C09106=1048.960,293.791,392.454,172.362,38.885,157.388
C09107=1048.967,294.039,392.422,172.365,38.887,157.388
C09108=1048.973,294.287,392.390,172.369,38.891,157.389
C09109=1048.980,294.535,392.357,172.372,38.894,157.390
C09110=1048.986,294.783,392.325,172.375,38.897,157.391
C09111=1048.993,295.030,392.293,172.379,38.900,157.392
C09112=1048.999,295.279,392.261,172.382,38.903,157.392
C09113=1049.006,295.526,392.229,172.385,38.906,157.393
C09114=1049.012,295.774,392.197,172.389,38.910,157.394
C09115=1049.019,296.021,392.165,172.392,38.913,157.395
C09116=1049.026,296.270,392.132,172.396,38.916,157.396
C09117=1049.032,296.518,392.100,172.398,38.919,157.396
C09118=1049.039,296.765,392.067,172.402,38.923,157.397
C09119=1049.046,297.013,392.035,172.406,38.925,157.398
C09120=1049.052,297.260,392.002,172.408,38.929,157.399
C09121=1049.058,297.509,391.970,172.412,38.932,157.400
C09122=1049.064,297.756,391.937,172.416,38.936,157.401
C09123=1049.071,298.003,391.905,172.419,38.939,157.401
C09124=1049.078,298.252,391.872,172.423,38.942,157.402
C09125=1049.084,298.499,391.839,172.425,38.945,157.403
C09126=1049.090,298.748,391.807,172.429,38.949,157.404
C09127=1049.097,298.995,391.774,172.433,38.952,157.405
C09128=1049.104,299.242,391.742,172.435,38.955,157.405
C09129=1049.110,299.490,391.710,172.439,38.959,157.406
C09130=1049.117,299.738,391.676,172.443,38.961,157.407
C09131=1049.123,299.986,391.644,172.446,38.965,157.408
C09132=1049.129,300.233,391.611,172.449,38.968,157.409
C09133=1049.136,300.481,391.579,172.453,38.971,157.410
C09134=1049.143,300.729,391.546,172.457,38.975,157.410
C09135=1049.150,300.977,391.513,172.460,38.978,157.411
C09136=1049.156,301.224,391.480,172.464,38.982,157.412
C09137=1049.162,301.472,391.447,172.467,38.984,157.413
C09138=1049.169,301.720,391.414,172.470,38.988,157.414
C09139=1049.176,301.967,391.382,172.474,38.991,157.414
C09140=1049.182,302.215,391.349,172.478,38.994,157.415
C09141=1049.189,302.463,391.317,172.481,38.998,157.416
C09142=1049.196,302.711,391.284,172.484,39.001,157.417
C09143=1049.202,302.958,391.251,172.488,39.004,157.418
C09144=1049.208,303.206,391.218,172.492,39.008,157.419
C09145=1049.216,303.454,391.186,172.494,39.011,157.419
C09146=1049.222,303.702,391.153,172.498,39.014,157.420
C09147=1049.229,303.949,391.119,172.502,39.017,157.421
C09148=1049.236,304.197,391.086,172.506,39.021,157.422
C09149=1049.244,304.491,391.047,172.510,39.024,157.423
C09150=1049.251,304.784,391.009,172.513,39.028,157.424
C09151=1049.259,305.078,390.970,172.518,39.032,157.425
C09152=1049.267,305.373,390.930,172.522,39.036,157.426
C09153=1049.274,305.620,390.898,172.526,39.040,157.427
C09154=1049.281,305.867,390.865,172.529,39.043,157.428
C09155=1049.288,306.115,390.831,172.533,39.046,157.428
C09156=1049.294,306.363,390.798,172.536,39.050,157.429
C09157=1049.301,306.611,390.765,172.540,39.053,157.430
C09158=1049.307,306.858,390.732,172.544,39.056,157.431
C09159=1049.314,307.106,390.699,172.547,39.060,157.432
C09160=1049.321,307.354,390.666,172.551,39.063,157.433
C09161=1049.328,307.601,390.632,172.554,39.066,157.434
C09162=1049.335,307.849,390.600,172.558,39.070,157.434
C09163=1049.342,308.096,390.566,172.562,39.073,157.435
C09164=1049.348,308.344,390.533,172.566,39.076,157.436
C09165=1049.355,308.592,390.500,172.568,39.080,157.437
C09166=1049.362,308.839,390.467,172.572,39.083,157.438
C09167=1049.369,309.088,390.434,172.576,39.086,157.439
C09168=1049.375,309.335,390.400,172.580,39.090,157.440
C09169=1049.382,309.583,390.367,172.584,39.093,157.440
C09170=1049.389,309.830,390.334,172.587,39.096,157.441
C09171=1049.396,310.078,390.301,172.591,39.100,157.442
C09172=1049.403,310.325,390.268,172.594,39.103,157.443
C09173=1049.410,310.573,390.235,172.598,39.106,157.444
C09174=1049.417,310.821,390.201,172.602,39.110,157.445
C09175=1049.424,311.068,390.167,172.605,39.113,157.445
C09176=1049.431,311.316,390.134,172.609,39.116,157.446
C09177=1049.437,311.563,390.101,172.613,39.119,157.447
C09178=1049.444,311.811,390.068,172.617,39.123,157.448
C09179=1049.451,312.059,390.034,172.621,39.126,157.449
C09180=1049.458,312.306,390.000,172.624,39.129,157.450
C09181=1049.465,312.554,389.967,172.628,39.133,157.451
C09182=1049.472,312.802,389.933,172.631,39.137,157.452
C09183=1049.479,313.049,389.900,172.635,39.140,157.452
C09184=1049.485,313.297,389.866,172.639,39.143,157.453
C09185=1049.492,313.545,389.832,172.643,39.147,157.454
C09186=1049.499,313.792,389.799,172.646,39.150,157.455
C09187=1049.505,314.040,389.765,172.650,39.154,157.456
C09188=1049.512,314.287,389.731,172.654,39.158,157.457
C09189=1049.518,314.535,389.697,172.658,39.161,157.458
C09190=1049.525,314.783,389.663,172.661,39.164,157.459
C09191=1049.531,315.030,389.629,172.665,39.168,157.460
C09192=1049.538,315.278,389.595,172.669,39.172,157.461
C09193=1049.544,315.525,389.561,172.672,39.175,157.462
C09194=1049.551,315.773,389.527,172.676,39.179,157.462
C09195=1049.558,316.021,389.493,172.680,39.183,157.463
C09196=1049.565,316.268,389.459,172.684,39.186,157.464
C09197=1049.571,316.516,389.425,172.688,39.189,157.465
C09198=1049.578,316.763,389.391,172.692,39.193,157.466
C09199=1049.584,317.011,389.357,172.696,39.196,157.467
C09200=1049.592,317.258,389.322,172.699,39.200,157.468
C09201=1049.598,317.506,389.288,172.703,39.204,157.469
C09202=1049.605,317.753,389.254,172.707,39.207,157.470
C09203=1049.611,318.001,389.220,172.711,39.211,157.471
C09204=1049.618,318.248,389.186,172.714,39.215,157.472
C09205=1049.626,318.546,389.145,172.719,39.219,157.473
C09206=1049.634,318.845,389.103,172.724,39.223,157.474
C09207=1049.642,319.143,389.062,172.728,39.227,157.475
C09208=1049.650,319.441,389.022,172.733,39.232,157.476
C09209=1049.657,319.689,388.986,172.737,39.236,157.477
C09210=1049.664,319.937,388.953,172.741,39.239,157.478
C09211=1049.671,320.185,388.918,172.745,39.243,157.479
C09212=1049.678,320.432,388.884,172.749,39.246,157.480
C09213=1049.684,320.679,388.850,172.753,39.250,157.481
C09214=1049.691,320.927,388.815,172.756,39.253,157.482
C09215=1049.698,321.174,388.781,172.760,39.257,157.483
C09216=1049.705,321.422,388.746,172.764,39.260,157.484
C09217=1049.712,321.670,388.712,172.768,39.264,157.485
C09218=1049.719,321.917,388.677,172.772,39.268,157.486
C09219=1049.726,322.165,388.643,172.776,39.271,157.486
C09220=1049.733,322.412,388.608,172.780,39.275,157.487
C09221=1049.739,322.660,388.574,172.784,39.279,157.488
C09222=1049.746,322.906,388.540,172.788,39.282,157.489
C09223=1049.752,323.154,388.505,172.792,39.286,157.490
C09224=1049.760,323.401,388.471,172.795,39.290,157.491
C09225=1049.766,323.649,388.436,172.799,39.293,157.492
C09226=1049.773,323.897,388.401,172.803,39.297,157.493
C09227=1049.780,324.144,388.367,172.807,39.301,157.494
C09228=1049.787,324.392,388.332,172.811,39.304,157.495
C09229=1049.794,324.639,388.298,172.816,39.308,157.496
C09230=1049.801,324.887,388.263,172.820,39.312,157.497
C09231=1049.808,325.134,388.228,172.824,39.315,157.498
C09232=1049.815,325.382,388.194,172.828,39.319,157.499
C09233=1049.822,325.630,388.159,172.832,39.323,157.500
C09234=1049.830,325.877,388.124,172.836,39.326,157.501
C09235=1049.836,326.125,388.090,172.840,39.330,157.502
C09236=1049.843,326.372,388.055,172.844,39.334,157.503
C09237=1049.851,326.619,388.020,172.847,39.337,157.504
C09238=1049.857,326.867,387.986,172.852,39.341,157.505
C09239=1049.864,327.115,387.951,172.856,39.345,157.506
C09240=1049.871,327.362,387.916,172.860,39.349,157.507
C09241=1049.878,327.609,387.881,172.864,39.352,157.508
C09242=1049.886,327.856,387.846,172.868,39.356,157.509
C09243=1049.893,328.105,387.812,172.872,39.360,157.510
C09244=1049.900,328.352,387.776,172.876,39.364,157.511
C09245=1049.907,328.599,387.742,172.881,39.367,157.512
C09246=1049.914,328.847,387.707,172.885,39.371,157.513
C09247=1049.921,329.094,387.672,172.889,39.375,157.514
C09248=1049.929,329.342,387.637,172.893,39.378,157.515
C09249=1049.935,329.589,387.602,172.897,39.382,157.516
C09250=1049.942,329.836,387.566,172.902,39.386,157.517
C09251=1049.949,330.084,387.531,172.906,39.390,157.518
C09252=1049.956,330.331,387.496,172.910,39.394,157.519
C09253=1049.963,330.579,387.461,172.914,39.398,157.520
C09254=1049.970,330.827,387.426,172.918,39.401,157.521
C09255=1049.977,331.074,387.390,172.922,39.405,157.522
C09256=1049.983,331.321,387.355,172.926,39.409,157.523
C09257=1049.991,331.568,387.319,172.931,39.413,157.524
C09258=1049.997,331.815,387.284,172.935,39.417,157.525
C09259=1050.005,332.064,387.249,172.939,39.421,157.526
C09260=1050.011,332.311,387.214,172.943,39.425,157.527
C09261=1050.019,332.604,387.171,172.948,39.429,157.528
C09262=1050.028,332.897,387.130,172.953,39.434,157.529
C09263=1050.036,333.191,387.087,172.958,39.439,157.530
C09264=1050.044,333.483,387.045,172.963,39.443,157.532
C09265=1050.051,333.731,387.010,172.967,39.447,157.533
C09266=1050.058,333.978,386.975,172.971,39.451,157.534
C09267=1050.066,334.225,386.939,172.975,39.456,157.535
C09268=1050.072,334.473,386.904,172.980,39.459,157.536
C09269=1050.079,334.720,386.868,172.984,39.463,157.537
C09270=1050.086,334.968,386.832,172.988,39.467,157.538
C09271=1050.093,335.215,386.796,172.992,39.471,157.539
C09272=1050.100,335.462,386.761,172.997,39.475,157.540
C09273=1050.107,335.710,386.725,173.001,39.479,157.541
C09274=1050.114,335.957,386.689,173.005,39.483,157.542
C09275=1050.122,336.205,386.654,173.011,39.487,157.543
C09276=1050.129,336.452,386.618,173.015,39.491,157.544
C09277=1050.135,336.699,386.582,173.019,39.495,157.546
C09278=1050.143,336.947,386.546,173.023,39.499,157.547
C09279=1050.150,337.194,386.510,173.028,39.503,157.548
C09280=1050.156,337.441,386.474,173.032,39.507,157.549
C09281=1050.163,337.689,386.438,173.036,39.511,157.550
C09282=1050.170,337.935,386.402,173.041,39.515,157.551
C09283=1050.177,338.184,386.366,173.045,39.519,157.552
C09284=1050.184,338.431,386.330,173.049,39.524,157.553
C09285=1050.192,338.678,386.294,173.054,39.527,157.554
C09286=1050.198,338.925,386.258,173.058,39.532,157.555
C09287=1050.205,339.172,386.223,173.062,39.536,157.556
C09288=1050.213,339.420,386.186,173.067,39.540,157.557
C09289=1050.219,339.667,386.150,173.071,39.544,157.558
C09290=1050.227,339.914,386.114,173.075,39.548,157.560
C09291=1050.234,340.161,386.078,173.081,39.552,157.561
C09292=1050.241,340.409,386.041,173.085,39.556,157.562
C09293=1050.247,340.656,386.006,173.089,39.561,157.563
C09294=1050.255,340.904,385.970,173.094,39.564,157.564
C09295=1050.261,341.151,385.933,173.098,39.569,157.565
C09296=1050.269,341.398,385.897,173.102,39.573,157.566
C09297=1050.277,341.646,385.861,173.107,39.577,157.567
C09298=1050.283,341.893,385.824,173.111,39.581,157.569
C09299=1050.291,342.140,385.788,173.116,39.585,157.570
C09300=1050.298,342.387,385.752,173.120,39.589,157.571
C09301=1050.305,342.635,385.715,173.124,39.594,157.572
C09302=1050.312,342.882,385.679,173.130,39.598,157.573
C09303=1050.319,343.128,385.642,173.134,39.602,157.574
C09304=1050.326,343.376,385.605,173.139,39.607,157.575
C09305=1050.333,343.623,385.569,173.143,39.610,157.576
C09306=1050.340,343.871,385.533,173.148,39.615,157.578
C09307=1050.348,344.118,385.496,173.152,39.619,157.579
C09308=1050.354,344.365,385.460,173.156,39.623,157.580
C09309=1050.361,344.612,385.422,173.161,39.628,157.581
C09310=1050.368,344.859,385.387,173.166,39.632,157.582
C09311=1050.375,345.107,385.350,173.171,39.636,157.583
C09312=1050.383,345.354,385.313,173.175,39.641,157.585
C09313=1050.390,345.601,385.276,173.180,39.645,157.586
C09314=1050.397,345.849,385.240,173.184,39.649,157.587
C09315=1050.405,346.095,385.203,173.189,39.654,157.588
C09316=1050.411,346.343,385.166,173.194,39.658,157.589
C09317=1050.419,346.632,385.123,173.199,39.663,157.591
C09318=1050.428,346.921,385.080,173.204,39.668,157.592
C09319=1050.437,347.211,385.037,173.210,39.673,157.593
C09320=1050.445,347.499,384.994,173.215,39.678,157.595
C09321=1050.452,347.747,384.957,173.220,39.682,157.596
C09322=1050.459,347.994,384.919,173.224,39.687,157.597
C09323=1050.467,348.242,384.883,173.230,39.692,157.598
C09324=1050.473,348.488,384.846,173.234,39.696,157.600
C09325=1050.480,348.735,384.808,173.239,39.700,157.601
C09326=1050.488,348.983,384.772,173.243,39.705,157.602
C09327=1050.495,349.230,384.735,173.248,39.709,157.603
C09328=1050.503,349.477,384.697,173.254,39.714,157.604
C09329=1050.510,349.725,384.660,173.258,39.718,157.606
C09330=1050.517,349.971,384.624,173.263,39.722,157.607
C09331=1050.524,350.218,384.586,173.267,39.727,157.608
C09332=1050.531,350.466,384.549,173.272,39.731,157.609
C09333=1050.538,350.713,384.512,173.277,39.736,157.610
C09334=1050.546,350.960,384.474,173.282,39.740,157.612
C09335=1050.554,351.207,384.437,173.287,39.745,157.613
C09336=1050.561,351.454,384.400,173.291,39.749,157.614
C09337=1050.568,351.701,384.362,173.296,39.754,157.615
C09338=1050.575,351.948,384.325,173.301,39.758,157.617
C09339=1050.582,352.195,384.288,173.306,39.763,157.618
C09340=1050.589,352.442,384.250,173.310,39.768,157.619
C09341=1050.596,352.690,384.213,173.315,39.772,157.620
C09342=1050.604,352.936,384.175,173.321,39.777,157.622
C09343=1050.611,353.183,384.137,173.325,39.781,157.623
C09344=1050.618,353.430,384.100,173.330,39.786,157.624
C09345=1050.625,353.677,384.062,173.336,39.790,157.625
C09346=1050.633,353.925,384.025,173.340,39.795,157.627
C09347=1050.640,354.172,383.987,173.345,39.799,157.628
C09348=1050.647,354.419,383.950,173.349,39.804,157.629
C09349=1050.654,354.666,383.912,173.355,39.809,157.631
C09350=1050.662,354.913,383.875,173.360,39.813,157.632
C09351=1050.669,355.160,383.837,173.364,39.818,157.633
C09352=1050.676,355.407,383.799,173.370,39.823,157.634
C09353=1050.684,355.654,383.761,173.375,39.827,157.636
C09354=1050.691,355.901,383.724,173.379,39.832,157.637
C09355=1050.698,356.148,383.686,173.384,39.837,157.638
C09356=1050.706,356.395,383.648,173.390,39.841,157.639
C09357=1050.714,356.643,383.610,173.395,39.846,157.641
C09358=1050.721,356.889,383.572,173.399,39.851,157.642
C09359=1050.728,357.136,383.535,173.405,39.856,157.643
C09360=1050.736,357.383,383.497,173.410,39.860,157.645
C09361=1050.743,357.630,383.459,173.414,39.865,157.646
C09362=1050.750,357.877,383.421,173.420,39.870,157.647
C09363=1050.757,358.124,383.382,173.425,39.874,157.649
C09364=1050.765,358.372,383.345,173.430,39.879,157.650
C09365=1050.773,358.618,383.306,173.435,39.884,157.651
C09366=1050.780,358.865,383.269,173.440,39.889,157.653
C09367=1050.787,359.112,383.230,173.445,39.894,157.654
C09368=1050.794,359.359,383.192,173.451,39.898,157.655
C09369=1050.801,359.606,383.154,173.455,39.903,157.657
C09370=1050.810,359.853,383.116,173.460,39.908,157.658
C09371=1050.817,360.099,383.077,173.466,39.913,157.659
C09372=1050.824,360.347,383.039,173.471,39.918,157.661
C09373=1050.833,360.641,382.993,173.477,39.924,157.662
C09374=1050.842,360.936,382.948,173.483,39.930,157.664
C09375=1050.851,361.230,382.902,173.489,39.935,157.666
C09376=1050.860,361.525,382.856,173.496,39.941,157.667
C09377=1050.867,361.771,382.818,173.501,39.946,157.669
C09378=1050.874,362.019,382.779,173.506,39.951,157.670
C09379=1050.882,362.266,382.741,173.511,39.956,157.671
C09380=1050.890,362.512,382.703,173.516,39.961,157.673
C09381=1050.897,362.760,382.664,173.522,39.966,157.674
C09382=1050.904,363.006,382.626,173.527,39.971,157.675
C09383=1050.912,363.253,382.587,173.533,39.976,157.677
C09384=1050.919,363.500,382.548,173.537,39.981,157.678
C09385=1050.927,363.747,382.510,173.543,39.986,157.680
C09386=1050.934,363.994,382.471,173.548,39.991,157.681
C09387=1050.942,364.240,382.432,173.553,39.996,157.683
C09388=1050.949,364.487,382.393,173.559,40.001,157.684
C09389=1050.957,364.734,382.355,173.564,40.006,157.685
C09390=1050.964,364.981,382.315,173.570,40.011,157.687
C09391=1050.971,365.228,382.277,173.575,40.016,157.688
C09392=1050.979,365.475,382.237,173.580,40.021,157.690
C09393=1050.986,365.721,382.198,173.585,40.027,157.691
C09394=1050.994,365.969,382.160,173.591,40.032,157.693
C09395=1051.001,366.216,382.121,173.596,40.037,157.694
C09396=1051.009,366.461,382.082,173.602,40.042,157.695
C09397=1051.016,366.709,382.043,173.607,40.047,157.697
C09398=1051.024,366.955,382.005,173.613,40.052,157.698
C09399=1051.032,367.202,381.965,173.618,40.058,157.700
C09400=1051.038,367.449,381.926,173.624,40.063,157.701
C09401=1051.047,367.696,381.886,173.629,40.068,157.703
C09402=1051.054,367.943,381.847,173.635,40.073,157.704
C09403=1051.062,368.189,381.808,173.640,40.078,157.706
C09404=1051.070,368.437,381.769,173.646,40.084,157.707
C09405=1051.077,368.683,381.730,173.651,40.089,157.709
C09406=1051.085,368.930,381.691,173.657,40.094,157.710
C09407=1051.092,369.176,381.651,173.662,40.099,157.712
C09408=1051.100,369.423,381.612,173.668,40.104,157.713
C09409=1051.108,369.670,381.573,173.673,40.110,157.715
C09410=1051.115,369.917,381.533,173.679,40.115,157.716
C09411=1051.123,370.163,381.494,173.684,40.120,157.718
C09412=1051.131,370.411,381.455,173.690,40.125,157.719
C09413=1051.139,370.657,381.416,173.696,40.131,157.721
C09414=1051.146,370.904,381.376,173.701,40.136,157.722
C09415=1051.154,371.150,381.336,173.707,40.141,157.724
C09416=1051.162,371.398,381.297,173.712,40.147,157.725
C09417=1051.169,371.644,381.258,173.718,40.153,157.727
C09418=1051.177,371.891,381.218,173.724,40.158,157.728
C09419=1051.185,372.138,381.178,173.729,40.163,157.730
C09420=1051.192,372.384,381.138,173.735,40.168,157.731
C09421=1051.200,372.631,381.098,173.740,40.174,157.733
C09422=1051.207,372.878,381.059,173.746,40.180,157.734
C09423=1051.214,373.124,381.019,173.753,40.185,157.736
C09424=1051.223,373.371,380.980,173.758,40.191,157.738
C09425=1051.231,373.617,380.940,173.764,40.196,157.739
C09426=1051.239,373.864,380.899,173.770,40.202,157.741
C09427=1051.246,374.111,380.859,173.775,40.207,157.742
C09428=1051.254,374.357,380.820,173.781,40.213,157.744
C09429=1051.264,374.670,380.768,173.788,40.220,157.746
C09430=1051.273,374.985,380.718,173.796,40.227,157.748
C09431=1051.283,375.297,380.667,173.803,40.234,157.750
C09432=1051.293,375.611,380.616,173.810,40.241,157.752
C09433=1051.301,375.858,380.576,173.816,40.247,157.754
C09434=1051.308,376.105,380.536,173.823,40.252,157.755
C09435=1051.317,376.351,380.495,173.828,40.258,157.757
C09436=1051.324,376.598,380.455,173.834,40.264,157.758
C09437=1051.332,376.844,380.415,173.840,40.269,157.760
C09438=1051.340,377.091,380.375,173.846,40.275,157.762
C09439=1051.348,377.337,380.334,173.852,40.280,157.763
C09440=1051.356,377.584,380.294,173.858,40.286,157.765
C09441=1051.363,377.830,380.254,173.864,40.292,157.767
C09442=1051.371,378.077,380.214,173.870,40.298,157.768
C09443=1051.379,378.324,380.173,173.876,40.304,157.770
C09444=1051.387,378.571,380.133,173.882,40.309,157.772
C09445=1051.395,378.817,380.093,173.888,40.315,157.773
C09446=1051.403,379.063,380.052,173.893,40.320,157.775
C09447=1051.411,379.310,380.012,173.900,40.326,157.777
C09448=1051.419,379.556,379.971,173.906,40.332,157.778
C09449=1051.427,379.803,379.931,173.912,40.338,157.780
C09450=1051.435,380.049,379.890,173.919,40.344,157.782
C09451=1051.443,380.295,379.850,173.924,40.350,157.783
C09452=1051.450,380.542,379.809,173.930,40.356,157.785
C09453=1051.458,380.789,379.768,173.936,40.361,157.787
C09454=1051.466,381.035,379.728,173.943,40.368,157.789
C09455=1051.473,381.282,379.687,173.949,40.374,157.790
C09456=1051.482,381.529,379.646,173.954,40.379,157.792
C09457=1051.490,381.775,379.605,173.961,40.386,157.794
C09458=1051.498,382.021,379.563,173.967,40.391,157.795
C09459=1051.506,382.267,379.522,173.973,40.397,157.797
C09460=1051.514,382.513,379.482,173.980,40.403,157.799
C09461=1051.521,382.760,379.440,173.986,40.409,157.801
C09462=1051.530,383.007,379.399,173.992,40.416,157.802
C09463=1051.538,383.253,379.359,173.998,40.421,157.804
C09464=1051.545,383.500,379.318,174.004,40.428,157.806
C09465=1051.553,383.746,379.276,174.011,40.433,157.808
C09466=1051.561,383.992,379.236,174.017,40.440,157.809
C09467=1051.569,384.239,379.194,174.024,40.446,157.811
C09468=1051.578,384.485,379.153,174.030,40.452,157.813
C09469=1051.586,384.731,379.112,174.036,40.458,157.815
C09470=1051.593,384.978,379.070,174.043,40.464,157.817
C09471=1051.602,385.224,379.029,174.049,40.471,157.818
C09472=1051.610,385.470,378.988,174.056,40.476,157.820
C09473=1051.618,385.717,378.946,174.062,40.483,157.822
C09474=1051.626,385.963,378.906,174.069,40.489,157.824
C09475=1051.634,386.210,378.863,174.075,40.495,157.826
C09476=1051.642,386.456,378.823,174.082,40.501,157.828
C09477=1051.651,386.702,378.781,174.087,40.508,157.829
C09478=1051.659,386.949,378.739,174.094,40.514,157.831
C09479=1051.667,387.195,378.698,174.100,40.520,157.833
C09480=1051.675,387.442,378.656,174.107,40.526,157.835
C09481=1051.683,387.687,378.615,174.113,40.533,157.837
C09482=1051.692,387.934,378.574,174.120,40.539,157.839
C09483=1051.700,388.180,378.532,174.126,40.545,157.840
C09484=1051.708,388.427,378.490,174.133,40.551,157.842
C09485=1051.719,388.772,378.432,174.142,40.560,157.845
C09486=1051.732,389.118,378.373,174.152,40.569,157.848
C09487=1051.743,389.465,378.314,174.161,40.578,157.850
C09488=1051.755,389.810,378.256,174.171,40.587,157.853
C09489=1051.763,390.056,378.213,174.177,40.594,157.855
C09490=1051.771,390.303,378.171,174.184,40.600,157.857
C09491=1051.779,390.549,378.130,174.191,40.607,157.859
C09492=1051.788,390.795,378.087,174.197,40.613,157.861
C09493=1051.795,391.041,378.045,174.204,40.620,157.862
C09494=1051.804,391.288,378.004,174.211,40.626,157.865
C09495=1051.813,391.534,377.961,174.218,40.633,157.866
C09496=1051.820,391.780,377.919,174.225,40.639,157.868
C09497=1051.829,392.026,377.877,174.232,40.646,157.870
C09498=1051.837,392.273,377.835,174.238,40.653,157.872
C09499=1051.846,392.519,377.792,174.245,40.659,157.874
C09500=1051.853,392.765,377.750,174.252,40.666,157.876
C09501=1051.862,393.011,377.708,174.259,40.673,157.878
C09502=1051.871,393.257,377.665,174.266,40.679,157.880
C09503=1051.878,393.503,377.623,174.273,40.686,157.882
C09504=1051.887,393.749,377.580,174.280,40.693,157.884
C09505=1051.895,393.996,377.538,174.286,40.700,157.886
C09506=1051.904,394.242,377.495,174.293,40.706,157.888
C09507=1051.913,394.488,377.452,174.301,40.713,157.890
C09508=1051.920,394.734,377.410,174.308,40.720,157.892
C09509=1051.929,394.980,377.367,174.315,40.726,157.894
C09510=1051.937,395.226,377.324,174.321,40.734,157.897
C09511=1051.946,395.472,377.282,174.329,40.741,157.899
C09512=1051.954,395.718,377.239,174.336,40.747,157.901
C09513=1051.963,395.965,377.196,174.343,40.754,157.903
C09514=1051.972,396.210,377.153,174.350,40.761,157.905
C09515=1051.980,396.457,377.111,174.358,40.768,157.907
C09516=1051.989,396.703,377.068,174.364,40.775,157.909
C09517=1051.997,396.949,377.025,174.371,40.782,157.911
C09518=1052.006,397.195,376.982,174.378,40.789,157.913
C09519=1052.013,397.441,376.938,174.386,40.796,157.915
C09520=1052.022,397.688,376.895,174.393,40.803,157.917
C09521=1052.030,397.934,376.852,174.400,40.810,157.919
C09522=1052.039,398.180,376.809,174.408,40.817,157.922
C09523=1052.047,398.426,376.766,174.415,40.824,157.924
C09524=1052.056,398.672,376.723,174.423,40.831,157.926
C09525=1052.065,398.917,376.679,174.429,40.838,157.928
C09526=1052.073,399.163,376.636,174.436,40.845,157.930
C09527=1052.082,399.409,376.593,174.444,40.853,157.932
C09528=1052.090,399.655,376.550,174.451,40.860,157.935
C09529=1052.100,399.901,376.506,174.459,40.867,157.937
C09530=1052.108,400.148,376.463,174.466,40.874,157.939
C09531=1052.117,400.394,376.420,174.474,40.881,157.941
C09532=1052.125,400.639,376.376,174.481,40.889,157.943
C09533=1052.133,400.885,376.333,174.488,40.896,157.946
C09534=1052.143,401.132,376.289,174.496,40.903,157.948
C09535=1052.151,401.378,376.246,174.503,40.910,157.950
C09536=1052.160,401.623,376.202,174.511,40.917,157.952
C09537=1052.168,401.870,376.158,174.519,40.925,157.954
C09538=1052.177,402.116,376.114,174.527,40.932,157.957
C09539=1052.186,402.362,376.071,174.534,40.939,157.959
C09540=1052.195,402.608,376.027,174.542,40.947,157.961
C09541=1052.207,402.971,375.962,174.553,40.958,157.964
C09542=1052.221,403.336,375.897,174.564,40.969,157.968
C09543=1052.233,403.700,375.832,174.575,40.980,157.971
C09544=1052.246,404.064,375.767,174.587,40.991,157.975
C09545=1052.255,404.310,375.723,174.595,40.999,157.977
C09546=1052.264,404.556,375.678,174.602,41.007,157.979
C09547=1052.272,404.802,375.635,174.611,41.014,157.982
C09548=1052.282,405.048,375.590,174.618,41.021,157.984
C09549=1052.290,405.294,375.546,174.626,41.029,157.986
C09550=1052.299,405.540,375.501,174.634,41.037,157.989
C09551=1052.307,405.785,375.458,174.641,41.045,157.991
C09552=1052.316,406.032,375.413,174.650,41.052,157.993
C09553=1052.325,406.277,375.368,174.658,41.060,157.996
C09554=1052.334,406.523,375.324,174.666,41.068,157.998
C09555=1052.343,406.769,375.280,174.673,41.076,158.001
C09556=1052.351,407.015,375.235,174.682,41.083,158.003
C09557=1052.360,407.261,375.190,174.690,41.091,158.005
C09558=1052.370,407.507,375.146,174.697,41.099,158.008
C09559=1052.378,407.752,375.101,174.706,41.107,158.010
C09560=1052.388,407.998,375.057,174.714,41.115,158.013
C09561=1052.396,408.244,375.011,174.722,41.123,158.015
C09562=1052.405,408.490,374.967,174.730,41.131,158.018
C09563=1052.414,408.735,374.922,174.738,41.138,158.020
C09564=1052.423,408.982,374.877,174.746,41.147,158.023
C09565=1052.433,409.227,374.833,174.755,41.154,158.025
C09566=1052.441,409.474,374.788,174.763,41.162,158.028
C09567=1052.450,409.719,374.743,174.772,41.170,158.030
C09568=1052.459,409.964,374.698,174.779,41.179,158.033
C09569=1052.468,410.210,374.653,174.787,41.186,158.035
C09570=1052.478,410.456,374.608,174.796,41.194,158.038
C09571=1052.487,410.702,374.563,174.804,41.203,158.040
C09572=1052.496,410.948,374.518,174.813,41.211,158.043
C09573=1052.505,411.194,374.473,174.821,41.219,158.045
C09574=1052.514,411.439,374.427,174.830,41.227,158.048
C09575=1052.523,411.685,374.382,174.839,41.235,158.050
C09576=1052.533,411.931,374.337,174.846,41.243,158.053
C09577=1052.542,412.177,374.292,174.856,41.252,158.056
C09578=1052.552,412.422,374.247,174.863,41.260,158.058
C09579=1052.561,412.668,374.201,174.872,41.268,158.061
C09580=1052.570,412.914,374.156,174.880,41.277,158.064
C09581=1052.580,413.159,374.111,174.889,41.285,158.066
C09582=1052.589,413.404,374.065,174.899,41.293,158.069
C09583=1052.598,413.650,374.020,174.906,41.301,158.071
C09584=1052.607,413.896,373.974,174.916,41.310,158.074
C09585=1052.617,414.142,373.928,174.925,41.318,158.077
C09586=1052.626,414.388,373.882,174.933,41.327,158.079
C09587=1052.635,414.633,373.836,174.942,41.335,158.082
C09588=1052.644,414.879,373.791,174.951,41.344,158.085
C09589=1052.653,415.124,373.745,174.959,41.352,158.088
C09590=1052.663,415.370,373.698,174.968,41.361,158.090
C09591=1052.672,415.616,373.653,174.977,41.369,158.093
C09592=1052.681,415.861,373.607,174.986,41.378,158.096
C09593=1052.691,416.106,373.560,174.995,41.387,158.098
C09594=1052.700,416.353,373.515,175.004,41.395,158.101
C09595=1052.709,416.598,373.469,175.013,41.404,158.104
C09596=1052.719,416.843,373.422,175.022,41.413,158.107
C09597=1052.733,417.218,373.352,175.036,41.426,158.111
C09598=1052.748,417.593,373.281,175.050,41.439,158.115
C09599=1052.762,417.968,373.211,175.064,41.452,158.120
C09600=1052.777,418.341,373.140,175.078,41.466,158.124
C09601=1052.787,418.587,373.093,175.087,41.475,158.127
C09602=1052.796,418.832,373.047,175.097,41.484,158.130
C09603=1052.806,419.078,373.001,175.106,41.493,158.132
C09604=1052.815,419.324,372.955,175.115,41.502,158.135
C09605=1052.825,419.570,372.907,175.125,41.511,158.138
C09606=1052.834,419.814,372.861,175.134,41.520,158.141
C09607=1052.844,420.060,372.814,175.144,41.529,158.144
C09608=1052.854,420.305,372.767,175.153,41.538,158.147
C09609=1052.863,420.551,372.720,175.163,41.547,158.150
C09610=1052.873,420.796,372.673,175.172,41.556,158.153
C09611=1052.882,421.042,372.627,175.181,41.565,158.156
C09612=1052.892,421.287,372.579,175.191,41.575,158.159
C09613=1052.902,421.532,372.532,175.200,41.584,158.162
C09614=1052.911,421.778,372.486,175.210,41.593,158.165
C09615=1052.921,422.023,372.438,175.219,41.602,158.168
C09616=1052.931,422.268,372.391,175.230,41.612,158.171
C09617=1052.941,422.514,372.343,175.240,41.621,158.174
C09618=1052.950,422.759,372.297,175.249,41.630,158.177
C09619=1052.960,423.005,372.249,175.259,41.640,158.180
C09620=1052.970,423.250,372.202,175.268,41.649,158.183
C09621=1052.979,423.493,372.155,175.279,41.658,158.186
C09622=1052.989,423.736,372.108,175.289,41.667,158.189
C09623=1052.999,423.980,372.061,175.298,41.677,158.192
C09624=1053.009,424.223,372.014,175.308,41.686,158.195
C09625=1053.019,424.466,371.967,175.319,41.696,158.199
C09626=1053.030,424.709,371.919,175.328,41.705,158.202
C09627=1053.039,424.952,371.872,175.338,41.715,158.205
C09628=1053.049,425.195,371.826,175.349,41.724,158.208
C09629=1053.058,425.441,371.778,175.358,41.733,158.211
C09630=1053.069,425.686,371.730,175.368,41.743,158.214
C09631=1053.078,425.931,371.682,175.379,41.753,158.218
C09632=1053.089,426.176,371.634,175.389,41.763,158.221
C09633=1053.099,426.422,371.586,175.400,41.773,158.224
C09634=1053.109,426.667,371.538,175.409,41.782,158.227
C09635=1053.119,426.912,371.490,175.420,41.792,158.230
C09636=1053.129,427.157,371.442,175.430,41.802,158.234
C09637=1053.139,427.402,371.394,175.441,41.812,158.237
C09638=1053.148,427.648,371.346,175.451,41.822,158.240
C09639=1053.159,427.892,371.298,175.462,41.831,158.243
C09640=1053.169,428.138,371.249,175.472,41.842,158.247
C09641=1053.179,428.383,371.201,175.483,41.852,158.250
C09642=1053.190,428.628,371.153,175.494,41.861,158.253
C09643=1053.199,428.872,371.104,175.504,41.872,158.257
C09644=1053.210,429.118,371.056,175.515,41.882,158.260
C09645=1053.220,429.363,371.007,175.526,41.891,158.264
C09646=1053.231,429.609,370.958,175.536,41.902,158.267
C09647=1053.241,429.853,370.910,175.547,41.912,158.270
C09648=1053.251,430.098,370.861,175.558,41.922,158.274
C09649=1053.262,430.343,370.812,175.569,41.932,158.277
C09650=1053.271,430.588,370.764,175.579,41.943,158.281
C09651=1053.282,430.833,370.714,175.591,41.953,158.284
C09652=1053.292,431.078,370.666,175.602,41.963,158.288
C09653=1053.309,431.470,370.587,175.619,41.980,158.293
C09654=1053.325,431.864,370.508,175.637,41.997,158.299
C09655=1053.342,432.256,370.430,175.655,42.014,158.305
C09656=1053.359,432.649,370.351,175.673,42.030,158.310
C09657=1053.369,432.894,370.301,175.684,42.041,158.314
C09658=1053.379,433.139,370.252,175.696,42.051,158.318
C09659=1053.390,433.384,370.202,175.707,42.062,158.321
C09660=1053.400,433.628,370.153,175.719,42.073,158.325
C09661=1053.412,433.873,370.104,175.730,42.084,158.329
C09662=1053.422,434.118,370.054,175.741,42.094,158.332
C09663=1053.433,434.363,370.005,175.754,42.105,158.336
C09664=1053.443,434.607,369.955,175.765,42.116,158.340
C09665=1053.454,434.853,369.906,175.777,42.126,158.343
C09666=1053.464,435.098,369.856,175.788,42.137,158.347
C09667=1053.475,435.342,369.806,175.800,42.148,158.351
C09668=1053.486,435.587,369.756,175.811,42.159,158.354
C09669=1053.497,435.832,369.707,175.824,42.170,158.358
C09670=1053.508,436.077,369.656,175.836,42.181,158.362
C09671=1053.518,436.322,369.607,175.847,42.192,158.366
C09672=1053.529,436.566,369.556,175.860,42.202,158.369
C09673=1053.541,436.811,369.507,175.872,42.214,158.373
C09674=1053.551,437.056,369.456,175.883,42.225,158.377
C09675=1053.562,437.300,369.406,175.896,42.236,158.381
C09676=1053.573,437.544,369.356,175.908,42.247,158.385
C09677=1053.583,437.789,369.306,175.920,42.259,158.389
C09678=1053.594,438.034,369.256,175.932,42.270,158.393
C09679=1053.605,438.278,369.206,175.944,42.281,158.397
C09680=1053.617,438.523,369.155,175.957,42.292,158.401
C09681=1053.627,438.768,369.104,175.969,42.304,158.405
C09682=1053.638,439.013,369.054,175.982,42.315,158.409
C09683=1053.649,439.256,369.003,175.994,42.327,158.413
C09684=1053.661,439.502,368.952,176.007,42.338,158.417
C09685=1053.671,439.746,368.901,176.020,42.349,158.421
C09686=1053.683,439.990,368.850,176.032,42.361,158.425
C09687=1053.694,440.234,368.800,176.045,42.372,158.429
C09688=1053.705,440.480,368.749,176.058,42.384,158.433
C09689=1053.716,440.724,368.697,176.070,42.396,158.437
C09690=1053.727,440.969,368.647,176.083,42.407,158.441
C09691=1053.738,441.213,368.596,176.096,42.419,158.445
C09692=1053.749,441.457,368.544,176.109,42.431,158.449
C09693=1053.761,441.702,368.493,176.121,42.443,158.454
C09694=1053.772,441.946,368.442,176.134,42.454,158.458
C09695=1053.783,442.191,368.390,176.148,42.466,158.462
C09696=1053.795,442.435,368.339,176.161,42.478,158.466
C09697=1053.806,442.679,368.288,176.174,42.490,158.471
C09698=1053.817,442.924,368.236,176.188,42.502,158.475
C09699=1053.829,443.168,368.184,176.201,42.514,158.479
C09700=1053.840,443.412,368.133,176.214,42.526,158.483
C09701=1053.852,443.657,368.081,176.228,42.538,158.488
C09702=1053.863,443.901,368.029,176.241,42.550,158.492
C09703=1053.874,444.145,367.978,176.255,42.563,158.496
C09704=1053.886,444.390,367.926,176.268,42.574,158.501
C09705=1053.898,444.634,367.873,176.281,42.587,158.505
C09706=1053.910,444.878,367.822,176.295,42.599,158.510
C09707=1053.921,445.122,367.769,176.310,42.611,158.514
C09708=1053.932,445.366,367.718,176.323,42.624,158.519
C09709=1053.945,445.612,367.666,176.337,42.636,158.523
C09710=1053.956,445.858,367.613,176.351,42.649,158.528
C09711=1053.967,446.104,367.560,176.365,42.661,158.532
C09712=1053.979,446.349,367.508,176.379,42.674,158.537
C09713=1053.992,446.592,367.456,176.394,42.686,158.541
C09714=1054.005,446.835,367.404,176.407,42.698,158.546
C09715=1054.018,447.079,367.354,176.422,42.711,158.550
C09716=1054.032,447.323,367.303,176.436,42.722,158.554
C09717=1054.048,447.567,367.254,176.450,42.734,158.559
C09718=1054.063,447.811,367.204,176.464,42.745,158.563
C09719=1054.080,448.055,367.157,176.480,42.757,158.567
C09720=1054.098,448.300,367.108,176.494,42.768,158.572
C09721=1054.116,448.544,367.060,176.508,42.779,158.576
C09722=1054.134,448.789,367.013,176.523,42.790,158.580
C09723=1054.154,449.034,366.967,176.538,42.800,158.584
C09724=1054.175,449.278,366.921,176.552,42.811,158.588
C09725=1054.196,449.524,366.876,176.568,42.821,158.592
C09726=1054.218,449.769,366.831,176.582,42.831,158.596
C09727=1054.241,450.015,366.787,176.598,42.841,158.600
C09728=1054.264,450.259,366.743,176.613,42.851,158.604
C09729=1053.943,450.280,366.451,176.612,42.951,158.633
C09730=1053.920,450.036,366.495,176.596,42.941,158.629
C09731=1053.897,449.790,366.539,176.582,42.931,158.625
C09732=1053.876,449.545,366.584,176.567,42.921,158.621
C09733=1053.854,449.299,366.629,176.551,42.911,158.617
C09734=1053.833,449.054,366.674,176.536,42.901,158.613
C09735=1053.813,448.810,366.721,176.521,42.890,158.608
C09736=1053.793,448.565,366.768,176.506,42.879,158.604
C09737=1053.776,448.320,366.815,176.492,42.868,158.600
C09738=1053.758,448.076,366.863,176.476,42.857,158.596
C09739=1053.742,447.831,366.912,176.462,42.846,158.591
C09740=1053.725,447.588,366.961,176.448,42.835,158.587
C09741=1053.710,447.344,367.010,176.433,42.823,158.583
C09742=1053.695,447.107,367.059,176.420,42.812,158.579
C09743=1053.682,446.871,367.108,176.405,42.800,158.574
C09744=1053.670,446.635,367.158,176.392,42.788,158.570
C09745=1053.658,446.400,367.208,176.378,42.777,158.566
C09746=1053.646,446.166,367.258,176.365,42.765,158.561
C09747=1053.635,445.932,367.308,176.351,42.752,158.557
C09748=1053.625,445.697,367.359,176.338,42.741,158.552
C09749=1053.613,445.463,367.408,176.324,42.729,158.548
C09750=1053.601,445.218,367.461,176.310,42.717,158.544
C09751=1053.590,444.974,367.512,176.296,42.704,158.539
C09752=1053.577,444.730,367.564,176.283,42.693,158.535
C09753=1053.566,444.486,367.617,176.269,42.680,158.530
C09754=1053.554,444.241,367.669,176.255,42.668,158.526
C09755=1053.543,443.996,367.721,176.241,42.656,158.522
C09756=1053.531,443.753,367.772,176.227,42.644,158.517
C09757=1053.520,443.508,367.824,176.214,42.632,158.513
C09758=1053.508,443.264,367.876,176.201,42.620,158.509
C09759=1053.496,443.019,367.927,176.187,42.608,158.504
C09760=1053.486,442.775,367.979,176.174,42.596,158.500
C09761=1053.474,442.531,368.030,176.161,42.584,158.496
C09762=1053.463,442.287,368.082,176.147,42.572,158.491
C09763=1053.452,442.042,368.133,176.134,42.560,158.487
C09764=1053.440,441.798,368.185,176.122,42.548,158.483
C09765=1053.429,441.553,368.236,176.108,42.537,158.479
C09766=1053.417,441.309,368.288,176.095,42.525,158.475
C09767=1053.406,441.065,368.338,176.082,42.514,158.470
C09768=1053.395,440.820,368.390,176.069,42.502,158.466
C09769=1053.384,440.576,368.441,176.056,42.491,158.462
C09770=1053.373,440.331,368.491,176.044,42.479,158.458
C09771=1053.361,440.087,368.543,176.031,42.467,158.454
C09772=1053.351,439.842,368.594,176.017,42.456,158.450
C09773=1053.340,439.598,368.644,176.006,42.445,158.446
C09774=1053.328,439.353,368.695,175.993,42.433,158.442
C09775=1053.317,439.109,368.746,175.980,42.422,158.438
C09776=1053.307,438.864,368.797,175.968,42.410,158.434
C09777=1053.295,438.619,368.847,175.955,42.399,158.430
C09778=1053.284,438.375,368.898,175.943,42.388,158.426
C09779=1053.273,438.130,368.948,175.930,42.376,158.422
C09780=1053.262,437.886,368.998,175.918,42.365,158.418
C09781=1053.251,437.641,369.049,175.905,42.354,158.414
C09782=1053.240,437.397,369.099,175.894,42.343,158.410
C09783=1053.230,437.152,369.150,175.882,42.332,158.406
C09784=1053.218,436.907,369.201,175.869,42.321,158.403
C09785=1053.208,436.662,369.250,175.857,42.310,158.399
C09786=1053.197,436.417,369.301,175.844,42.299,158.395
C09787=1053.186,436.172,369.350,175.833,42.288,158.391
C09788=1053.175,435.928,369.400,175.821,42.277,158.387
C09789=1053.164,435.683,369.449,175.809,42.266,158.383
C09790=1053.153,435.439,369.500,175.797,42.255,158.380
C09791=1053.142,435.194,369.549,175.785,42.244,158.376
C09792=1053.132,434.950,369.599,175.774,42.234,158.372
C09793=1053.121,434.705,369.649,175.762,42.223,158.369
C09794=1053.110,434.460,369.699,175.750,42.212,158.365
C09795=1053.100,434.215,369.748,175.738,42.202,158.361
C09796=1053.089,433.970,369.798,175.727,42.191,158.357
C09797=1053.078,433.725,369.847,175.715,42.180,158.354
C09798=1053.068,433.480,369.897,175.704,42.169,158.350
C09799=1053.057,433.236,369.946,175.692,42.159,158.346
C09800=1053.046,432.991,369.995,175.681,42.149,158.343
C09801=1053.036,432.746,370.045,175.670,42.138,158.339
C09802=1053.019,432.351,370.124,175.652,42.121,158.334
C09803=1053.002,431.957,370.204,175.633,42.104,158.328
C09804=1052.986,431.562,370.283,175.615,42.088,158.322
C09805=1052.969,431.166,370.362,175.597,42.071,158.316
C09806=1052.959,430.921,370.411,175.586,42.061,158.313
C09807=1052.949,430.676,370.460,175.574,42.050,158.309
C09808=1052.937,430.431,370.509,175.564,42.040,158.306
C09809=1052.928,430.187,370.557,175.553,42.030,158.302
C09810=1052.918,429.942,370.607,175.542,42.019,158.299
C09811=1052.907,429.697,370.655,175.531,42.010,158.296
C09812=1052.897,429.452,370.704,175.521,41.999,158.292
C09813=1052.886,429.206,370.752,175.510,41.989,158.289
C09814=1052.877,428.961,370.801,175.498,41.979,158.285
C09815=1052.866,428.717,370.849,175.487,41.969,158.282
C09816=1052.856,428.471,370.898,175.477,41.959,158.279
C09817=1052.846,428.226,370.946,175.466,41.950,158.275
C09818=1052.836,427.981,370.994,175.455,41.940,158.272
C09819=1052.826,427.736,371.043,175.445,41.929,158.269
C09820=1052.815,427.491,371.091,175.434,41.920,158.265
C09821=1052.805,427.246,371.139,175.425,41.910,158.262
C09822=1052.795,427.000,371.187,175.414,41.900,158.259
C09823=1052.785,426.756,371.235,175.404,41.890,158.256
C09824=1052.775,426.511,371.284,175.393,41.881,158.252
C09825=1052.765,426.265,371.331,175.383,41.871,158.249
C09826=1052.755,426.020,371.380,175.372,41.861,158.246
C09827=1052.744,425.774,371.427,175.362,41.851,158.243
C09828=1052.735,425.529,371.476,175.351,41.842,158.239
C09829=1052.724,425.284,371.523,175.342,41.833,158.236
C09830=1052.715,425.039,371.571,175.331,41.823,158.233
C09831=1052.705,424.794,371.618,175.321,41.813,158.230
C09832=1052.694,424.549,371.666,175.311,41.804,158.227
C09833=1052.685,424.303,371.714,175.301,41.795,158.224
C09834=1052.675,424.058,371.761,175.291,41.785,158.221
C09835=1052.665,423.812,371.808,175.281,41.776,158.217
C09836=1052.655,423.568,371.856,175.271,41.766,158.214
C09837=1052.645,423.322,371.904,175.261,41.757,158.211
C09838=1052.635,423.078,371.951,175.251,41.747,158.208
C09839=1052.626,422.832,371.998,175.241,41.739,158.205
C09840=1052.616,422.586,372.045,175.231,41.729,158.202
C09841=1052.605,422.341,372.092,175.221,41.720,158.199
C09842=1052.596,422.095,372.140,175.212,41.711,158.196
C09843=1052.586,421.851,372.187,175.202,41.701,158.193
C09844=1052.576,421.605,372.234,175.192,41.692,158.190
C09845=1052.567,421.359,372.281,175.182,41.683,158.187
C09846=1052.557,421.114,372.328,175.173,41.674,158.184
C09847=1052.547,420.869,372.375,175.163,41.665,158.181
C09848=1052.537,420.623,372.422,175.154,41.656,158.178
C09849=1052.529,420.379,372.469,175.144,41.646,158.175
C09850=1052.519,420.133,372.516,175.135,41.637,158.172
C09851=1052.508,419.887,372.563,175.125,41.628,158.169
C09852=1052.500,419.642,372.609,175.116,41.619,158.166
C09853=1052.490,419.397,372.657,175.106,41.610,158.163
C09854=1052.480,419.151,372.703,175.097,41.602,158.161
C09855=1052.471,418.905,372.749,175.088,41.593,158.158
C09856=1052.461,418.660,372.795,175.078,41.584,158.155
C09857=1052.451,418.414,372.842,175.069,41.575,158.152
C09858=1052.437,418.041,372.913,175.055,41.562,158.148
C09859=1052.422,417.670,372.982,175.041,41.548,158.143
C09860=1052.408,417.297,373.053,175.027,41.535,158.139
C09861=1052.393,416.924,373.123,175.013,41.522,158.135
C09862=1052.384,416.679,373.170,175.004,41.514,158.132
C09863=1052.375,416.433,373.216,174.994,41.505,158.129
C09864=1052.365,416.187,373.262,174.985,41.496,158.126
C09865=1052.356,415.942,373.308,174.977,41.487,158.124
C09866=1052.346,415.700,373.353,174.968,41.479,158.121
C09867=1052.337,415.459,373.399,174.959,41.471,158.118
C09868=1052.328,415.217,373.443,174.950,41.462,158.116
C09869=1052.319,414.975,373.490,174.941,41.454,158.113
C09870=1052.309,414.733,373.534,174.932,41.446,158.110
C09871=1052.300,414.491,373.579,174.924,41.437,158.107
C09872=1052.291,414.250,373.625,174.915,41.429,158.105
C09873=1052.282,414.008,373.669,174.906,41.420,158.102
C09874=1052.273,413.762,373.715,174.898,41.412,158.100
C09875=1052.264,413.517,373.761,174.889,41.404,158.097
C09876=1052.255,413.271,373.806,174.880,41.396,158.094
C09877=1052.245,413.025,373.852,174.872,41.387,158.092
C09878=1052.236,412.779,373.898,174.863,41.379,158.089
C09879=1052.226,412.534,373.943,174.854,41.371,158.086
C09880=1052.217,412.288,373.988,174.846,41.362,158.084
C09881=1052.208,412.042,374.034,174.837,41.354,158.081
C09882=1052.198,411.797,374.078,174.829,41.346,158.079
C09883=1052.189,411.551,374.124,174.820,41.338,158.076
C09884=1052.180,411.305,374.169,174.812,41.330,158.073
C09885=1052.171,411.060,374.214,174.803,41.322,158.071
C09886=1052.162,410.814,374.260,174.795,41.314,158.068
C09887=1052.152,410.568,374.304,174.786,41.306,158.066
C09888=1052.143,410.322,374.350,174.778,41.297,158.063
C09889=1052.134,410.076,374.395,174.769,41.290,158.061
C09890=1052.125,409.831,374.439,174.762,41.282,158.058
C09891=1052.116,409.585,374.485,174.753,41.274,158.056
C09892=1052.107,409.340,374.529,174.745,41.266,158.053
C09893=1052.098,409.093,374.574,174.736,41.258,158.051
C09894=1052.089,408.848,374.619,174.728,41.250,158.048
C09895=1052.079,408.602,374.664,174.719,41.242,158.046
C09896=1052.071,408.356,374.709,174.711,41.234,158.043
C09897=1052.061,408.111,374.753,174.704,41.226,158.041
C09898=1052.053,407.864,374.798,174.695,41.218,158.038
C09899=1052.044,407.619,374.843,174.687,41.211,158.036
C09900=1052.034,407.372,374.888,174.679,41.203,158.034
C09901=1052.026,407.127,374.933,174.670,41.195,158.031
C09902=1052.017,406.881,374.977,174.663,41.187,158.029
C09903=1052.009,406.635,375.021,174.655,41.180,158.026
C09904=1051.999,406.390,375.066,174.646,41.172,158.024
C09905=1051.990,406.143,375.111,174.639,41.164,158.021
C09906=1051.982,405.898,375.155,174.631,41.157,158.019
C09907=1051.973,405.652,375.199,174.623,41.149,158.017
C09908=1051.965,405.406,375.243,174.615,41.141,158.014
C09909=1051.955,405.160,375.288,174.607,41.134,158.012
C09910=1051.947,404.915,375.333,174.599,41.126,158.010
C09911=1051.937,404.668,375.377,174.591,41.118,158.007
C09912=1051.929,404.423,375.421,174.584,41.111,158.005
C09913=1051.920,404.177,375.465,174.575,41.104,158.003
C09914=1051.907,403.802,375.532,174.564,41.092,157.999
C09915=1051.894,403.429,375.598,174.552,41.080,157.995
C09916=1051.880,403.055,375.666,174.540,41.069,157.992
C09917=1051.867,402.681,375.732,174.528,41.058,157.989
C09918=1051.858,402.436,375.776,174.521,41.051,157.986
C09919=1051.849,402.189,375.819,174.513,41.044,157.984
C09920=1051.841,401.943,375.864,174.506,41.036,157.982
C09921=1051.832,401.698,375.907,174.498,41.029,157.980
C09922=1051.823,401.451,375.951,174.491,41.022,157.977
C09923=1051.814,401.206,375.995,174.483,41.014,157.975
C09924=1051.806,400.960,376.038,174.476,41.007,157.973
C09925=1051.796,400.713,376.082,174.468,41.000,157.971
C09926=1051.789,400.467,376.125,174.461,40.993,157.969
C09927=1051.780,400.221,376.168,174.454,40.986,157.966
C09928=1051.771,399.976,376.212,174.446,40.978,157.964
C09929=1051.762,399.729,376.255,174.439,40.971,157.962
C09930=1051.754,399.483,376.299,174.431,40.964,157.960
C09931=1051.745,399.237,376.342,174.424,40.957,157.958
C09932=1051.736,398.991,376.385,174.416,40.950,157.955
C09933=1051.728,398.745,376.428,174.409,40.943,157.953
C09934=1051.719,398.499,376.471,174.402,40.936,157.951
C09935=1051.711,398.254,376.515,174.394,40.928,157.949
C09936=1051.702,398.008,376.558,174.387,40.922,157.947
C09937=1051.693,397.761,376.601,174.379,40.915,157.945
C09938=1051.685,397.515,376.645,174.372,40.907,157.942
C09939=1051.677,397.268,376.688,174.365,40.901,157.940
C09940=1051.668,397.022,376.731,174.357,40.893,157.938
C09941=1051.660,396.776,376.774,174.350,40.887,157.936
C09942=1051.652,396.531,376.817,174.344,40.880,157.934
C09943=1051.643,396.284,376.860,174.336,40.873,157.932
C09944=1051.634,396.038,376.902,174.329,40.866,157.930
C09945=1051.626,395.793,376.945,174.322,40.859,157.928
C09946=1051.617,395.547,376.988,174.314,40.852,157.926
C09947=1051.609,395.300,377.031,174.307,40.845,157.924
C09948=1051.601,395.054,377.073,174.300,40.839,157.922
C09949=1051.592,394.808,377.116,174.294,40.832,157.920
C09950=1051.584,394.562,377.159,174.286,40.825,157.918
C09951=1051.575,394.315,377.201,174.279,40.819,157.916
C09952=1051.566,394.069,377.244,174.272,40.812,157.914
C09953=1051.558,393.824,377.286,174.266,40.805,157.912
C09954=1051.550,393.577,377.329,174.258,40.798,157.910
C09955=1051.542,393.331,377.372,174.251,40.792,157.907
C09956=1051.534,393.085,377.414,174.244,40.785,157.905
C09957=1051.525,392.839,377.456,174.238,40.778,157.903
C09958=1051.517,392.593,377.498,174.231,40.772,157.902
C09959=1051.509,392.346,377.541,174.223,40.765,157.900
C09960=1051.500,392.100,377.584,174.216,40.759,157.898
C09961=1051.492,391.854,377.625,174.210,40.752,157.896
C09962=1051.483,391.608,377.667,174.203,40.746,157.894
C09963=1051.475,391.361,377.710,174.196,40.739,157.892
C09964=1051.467,391.116,377.752,174.190,40.733,157.890
C09965=1051.458,390.869,377.794,174.183,40.726,157.888
C09966=1051.450,390.623,377.836,174.176,40.720,157.886
C09967=1051.442,390.377,377.878,174.169,40.713,157.884
C09968=1051.434,390.130,377.920,174.162,40.707,157.882
C09969=1051.426,389.884,377.962,174.155,40.700,157.880
C09970=1051.414,389.536,378.022,174.146,40.691,157.877
C09971=1051.402,389.189,378.081,174.136,40.682,157.875
C09972=1051.391,388.841,378.140,174.127,40.673,157.872
C09973=1051.379,388.493,378.199,174.117,40.664,157.869
C09974=1051.370,388.247,378.240,174.111,40.658,157.867
C09975=1051.362,388.000,378.282,174.104,40.651,157.866
C09976=1051.354,387.754,378.323,174.098,40.645,157.864
C09977=1051.346,387.507,378.366,174.091,40.639,157.862
C09978=1051.338,387.261,378.406,174.084,40.633,157.860
C09979=1051.329,387.015,378.448,174.078,40.626,157.858
C09980=1051.321,386.769,378.490,174.071,40.620,157.856
C09981=1051.313,386.523,378.531,174.065,40.614,157.854
C09982=1051.305,386.276,378.573,174.058,40.608,157.853
C09983=1051.296,386.030,378.614,174.052,40.602,157.851
C09984=1051.288,385.783,378.655,174.045,40.596,157.849
C09985=1051.280,385.537,378.697,174.039,40.589,157.847
C09986=1051.272,385.291,378.738,174.032,40.583,157.845
C09987=1051.263,385.045,378.780,174.027,40.577,157.844
C09988=1051.256,384.798,378.821,174.020,40.571,157.842
C09989=1051.248,384.552,378.861,174.014,40.565,157.840
C09990=1051.240,384.305,378.904,174.008,40.559,157.838
C09991=1051.232,384.059,378.944,174.001,40.553,157.836
C09992=1051.224,383.812,378.985,173.995,40.547,157.835
C09993=1051.216,383.566,379.027,173.988,40.541,157.833
C09994=1051.208,383.320,379.068,173.982,40.535,157.831
C09995=1051.199,383.073,379.109,173.975,40.529,157.829
C09996=1051.192,382.827,379.150,173.969,40.523,157.828
//INST
///DATE 2021/06/25 14:47
///ATTR SC,RW,RJ
////FRAME ROBOT
///GROUP1 RB1
NOP
MOVL C00000 V=800.0 PL=0
MOVL C00001 V=800.0 PL=0
MOVL C00002 V=800.0 PL=0
MOVL C00003 V=800.0 PL=0
MOVL C00004 V=800.0 PL=0
MOVL C00005 V=800.0 PL=0
MOVL C00006 V=800.0 PL=0
MOVL C00007 V=800.0 PL=0
MOVL C00008 V=800.0 PL=0
MOVL C00009 V=800.0 PL=0
MOVL C00010 V=800.0 PL=0
MOVL C00011 V=800.0 PL=0
MOVL C00012 V=800.0 PL=0
MOVL C00013 V=800.0 PL=0
MOVL C00014 V=800.0 PL=0
MOVL C00015 V=800.0 PL=0
MOVL C00016 V=800.0 PL=0
MOVL C00017 V=800.0 PL=0
MOVL C00018 V=800.0 PL=0
MOVL C00019 V=800.0 PL=0
MOVL C00020 V=800.0 PL=0
MOVL C00021 V=800.0 PL=0
MOVL C00022 V=800.0 PL=0
MOVL C00023 V=800.0 PL=0
MOVL C00024 V=800.0 PL=0
MOVL C00025 V=800.0 PL=0
MOVL C00026 V=800.0 PL=0
MOVL C00027 V=800.0 PL=0
MOVL C00028 V=800.0 PL=0
MOVL C00029 V=800.0 PL=0
MOVL C00030 V=800.0 PL=0
MOVL C00031 V=800.0 PL=0
MOVL C00032 V=800.0 PL=0
MOVL C00033 V=800.0 PL=0
MOVL C00034 V=800.0 PL=0
MOVL C00035 V=800.0 PL=0
MOVL C00036 V=800.0 PL=0
MOVL C00037 V=800.0 PL=0
MOVL C00038 V=800.0 PL=0
MOVL C00039 V=800.0 PL=0
MOVL C00040 V=800.0 PL=0
MOVL C00041 V=800.0 PL=0
MOVL C00042 V=800.0 PL=0
MOVL C00043 V=800.0 PL=0
MOVL C00044 V=800.0 PL=0
MOVL C00045 V=800.0 PL=0
MOVL C00046 V=800.0 PL=0
MOVL C00047 V=800.0 PL=0
MOVL C00048 V=800.0 PL=0
MOVL C00049 V=800.0 PL=0
MOVL C00050 V=800.0 PL=0
MOVL C00051 V=800.0 PL=0
MOVL C00052 V=800.0 PL=0
MOVL C00053 V=800.0 PL=0
MOVL C00054 V=800.0 PL=0
MOVL C00055 V=800.0 PL=0
MOVL C00056 V=800.0 PL=0
MOVL C00057 V=800.0 PL=0
MOVL C00058 V=800.0 PL=0
MOVL C00059 V=800.0 PL=0
MOVL C00060 V=800.0 PL=0
MOVL C00061 V=800.0 PL=0
MOVL C00062 V=800.0 PL=0
MOVL C00063 V=800.0 PL=0
MOVL C00064 V=800.0 PL=0
MOVL C00065 V=800.0 PL=0
MOVL C00066 V=800.0 PL=0
MOVL C00067 V=800.0 PL=0
MOVL C00068 V=800.0 PL=0
MOVL C00069 V=800.0 PL=0
MOVL C00070 V=800.0 PL=0
MOVL C00071 V=800.0 PL=0
MOVL C00072 V=800.0 PL=0
MOVL C00073 V=800.0 PL=0
MOVL C00074 V=800.0 PL=0
MOVL C00075 V=800.0 PL=0
MOVL C00076 V=800.0 PL=0
MOVL C00077 V=800.0 PL=0
MOVL C00078 V=800.0 PL=0
MOVL C00079 V=800.0 PL=0
MOVL C00080 V=800.0 PL=0
MOVL C00081 V=800.0 PL=0
MOVL C00082 V=800.0 PL=0
MOVL C00083 V=800.0 PL=0
MOVL C00084 V=800.0 PL=0
MOVL C00085 V=800.0 PL=0
MOVL C00086 V=800.0 PL=0
MOVL C00087 V=800.0 PL=0
MOVL C00088 V=800.0 PL=0
MOVL C00089 V=800.0 PL=0
MOVL C00090 V=800.0 PL=0
MOVL C00091 V=800.0 PL=0
MOVL C00092 V=800.0 PL=0
MOVL C00093 V=800.0 PL=0
MOVL C00094 V=800.0 PL=0
MOVL C00095 V=800.0 PL=0
MOVL C00096 V=800.0 PL=0
MOVL C00097 V=800.0 PL=0
MOVL C00098 V=800.0 PL=0
MOVL C00099 V=800.0 PL=0
MOVL C00100 V=800.0 PL=0
MOVL C00101 V=800.0 PL=0
MOVL C00102 V=800.0 PL=0
MOVL C00103 V=800.0 PL=0
MOVL C00104 V=800.0 PL=0
MOVL C00105 V=800.0 PL=0
MOVL C00106 V=800.0 PL=0
MOVL C00107 V=800.0 PL=0
MOVL C00108 V=800.0 PL=0
MOVL C00109 V=800.0 PL=0
MOVL C00110 V=800.0 PL=0
MOVL C00111 V=800.0 PL=0
MOVL C00112 V=800.0 PL=0
MOVL C00113 V=800.0 PL=0
MOVL C00114 V=800.0 PL=0
MOVL C00115 V=800.0 PL=0
MOVL C00116 V=800.0 PL=0
MOVL C00117 V=800.0 PL=0
MOVL C00118 V=800.0 PL=0
MOVL C00119 V=800.0 PL=0
MOVL C00120 V=800.0 PL=0
MOVL C00121 V=800.0 PL=0
MOVL C00122 V=800.0 PL=0
MOVL C00123 V=800.0 PL=0
MOVL C00124 V=800.0 PL=0
MOVL C00125 V=800.0 PL=0
MOVL C00126 V=800.0 PL=0
MOVL C00127 V=800.0 PL=0
MOVL C00128 V=800.0 PL=0
MOVL C00129 V=800.0 PL=0
MOVL C00130 V=800.0 PL=0
MOVL C00131 V=800.0 PL=0
MOVL C00132 V=800.0 PL=0
MOVL C00133 V=800.0 PL=0
MOVL C00134 V=800.0 PL=0
MOVL C00135 V=800.0 PL=0
MOVL C00136 V=800.0 PL=0
MOVL C00137 V=800.0 PL=0
MOVL C00138 V=800.0 PL=0
MOVL C00139 V=800.0 PL=0
MOVL C00140 V=800.0 PL=0
MOVL C00141 V=800.0 PL=0
MOVL C00142 V=800.0 PL=0
MOVL C00143 V=800.0 PL=0
MOVL C00144 V=800.0 PL=0
MOVL C00145 V=800.0 PL=0
MOVL C00146 V=800.0 PL=0
MOVL C00147 V=800.0 PL=0
MOVL C00148 V=800.0 PL=0
MOVL C00149 V=800.0 PL=0
MOVL C00150 V=800.0 PL=0
MOVL C00151 V=800.0 PL=0
MOVL C00152 V=800.0 PL=0
MOVL C00153 V=800.0 PL=0
MOVL C00154 V=800.0 PL=0
MOVL C00155 V=800.0 PL=0
MOVL C00156 V=800.0 PL=0
MOVL C00157 V=800.0 PL=0
MOVL C00158 V=800.0 PL=0
MOVL C00159 V=800.0 PL=0
MOVL C00160 V=800.0 PL=0
MOVL C00161 V=800.0 PL=0
MOVL C00162 V=800.0 PL=0
MOVL C00163 V=800.0 PL=0
MOVL C00164 V=800.0 PL=0
MOVL C00165 V=800.0 PL=0
MOVL C00166 V=800.0 PL=0
MOVL C00167 V=800.0 PL=0
MOVL C00168 V=800.0 PL=0
MOVL C00169 V=800.0 PL=0
MOVL C00170 V=800.0 PL=0
MOVL C00171 V=800.0 PL=0
MOVL C00172 V=800.0 PL=0
MOVL C00173 V=800.0 PL=0
MOVL C00174 V=800.0 PL=0
MOVL C00175 V=800.0 PL=0
MOVL C00176 V=800.0 PL=0
MOVL C00177 V=800.0 PL=0
MOVL C00178 V=800.0 PL=0
MOVL C00179 V=800.0 PL=0
MOVL C00180 V=800.0 PL=0
MOVL C00181 V=800.0 PL=0
MOVL C00182 V=800.0 PL=0
MOVL C00183 V=800.0 PL=0
MOVL C00184 V=800.0 PL=0
MOVL C00185 V=800.0 PL=0
MOVL C00186 V=800.0 PL=0
MOVL C00187 V=800.0 PL=0
MOVL C00188 V=800.0 PL=0
MOVL C00189 V=800.0 PL=0
MOVL C00190 V=800.0 PL=0
MOVL C00191 V=800.0 PL=0
MOVL C00192 V=800.0 PL=0
MOVL C00193 V=800.0 PL=0
MOVL C00194 V=800.0 PL=0
MOVL C00195 V=800.0 PL=0
MOVL C00196 V=800.0 PL=0
MOVL C00197 V=800.0 PL=0
MOVL C00198 V=800.0 PL=0
MOVL C00199 V=800.0 PL=0
MOVL C00200 V=800.0 PL=0
MOVL C00201 V=800.0 PL=0
MOVL C00202 V=800.0 PL=0
MOVL C00203 V=800.0 PL=0
MOVL C00204 V=800.0 PL=0
MOVL C00205 V=800.0 PL=0
MOVL C00206 V=800.0 PL=0
MOVL C00207 V=800.0 PL=0
MOVL C00208 V=800.0 PL=0
MOVL C00209 V=800.0 PL=0
MOVL C00210 V=800.0 PL=0
MOVL C00211 V=800.0 PL=0
MOVL C00212 V=800.0 PL=0
MOVL C00213 V=800.0 PL=0
MOVL C00214 V=800.0 PL=0
MOVL C00215 V=800.0 PL=0
MOVL C00216 V=800.0 PL=0
MOVL C00217 V=800.0 PL=0
MOVL C00218 V=800.0 PL=0
MOVL C00219 V=800.0 PL=0
MOVL C00220 V=800.0 PL=0
MOVL C00221 V=800.0 PL=0
MOVL C00222 V=800.0 PL=0
MOVL C00223 V=800.0 PL=0
MOVL C00224 V=800.0 PL=0
MOVL C00225 V=800.0 PL=0
MOVL C00226 V=800.0 PL=0
MOVL C00227 V=800.0 PL=0
MOVL C00228 V=800.0 PL=0
MOVL C00229 V=800.0 PL=0
MOVL C00230 V=800.0 PL=0
MOVL C00231 V=800.0 PL=0
MOVL C00232 V=800.0 PL=0
MOVL C00233 V=800.0 PL=0
MOVL C00234 V=800.0 PL=0
MOVL C00235 V=800.0 PL=0
MOVL C00236 V=800.0 PL=0
MOVL C00237 V=800.0 PL=0
MOVL C00238 V=800.0 PL=0
MOVL C00239 V=800.0 PL=0
MOVL C00240 V=800.0 PL=0
MOVL C00241 V=800.0 PL=0
MOVL C00242 V=800.0 PL=0
MOVL C00243 V=800.0 PL=0
MOVL C00244 V=800.0 PL=0
MOVL C00245 V=800.0 PL=0
MOVL C00246 V=800.0 PL=0
MOVL C00247 V=800.0 PL=0
MOVL C00248 V=800.0 PL=0
MOVL C00249 V=800.0 PL=0
MOVL C00250 V=800.0 PL=0
MOVL C00251 V=800.0 PL=0
MOVL C00252 V=800.0 PL=0
MOVL C00253 V=800.0 PL=0
MOVL C00254 V=800.0 PL=0
MOVL C00255 V=800.0 PL=0
MOVL C00256 V=800.0 PL=0
MOVL C00257 V=800.0 PL=0
MOVL C00258 V=800.0 PL=0
MOVL C00259 V=800.0 PL=0
MOVL C00260 V=800.0 PL=0
MOVL C00261 V=800.0 PL=0
MOVL C00262 V=800.0 PL=0
MOVL C00263 V=800.0 PL=0
MOVL C00264 V=800.0 PL=0
MOVL C00265 V=800.0 PL=0
MOVL C00266 V=800.0 PL=0
MOVL C00267 V=800.0 PL=0
MOVL C00268 V=800.0 PL=0
MOVL C00269 V=800.0 PL=0
MOVL C00270 V=800.0 PL=0
MOVL C00271 V=800.0 PL=0
MOVL C00272 V=800.0 PL=0
MOVL C00273 V=800.0 PL=0
MOVL C00274 V=800.0 PL=0
MOVL C00275 V=800.0 PL=0
MOVL C00276 V=800.0 PL=0
MOVL C00277 V=800.0 PL=0
MOVL C00278 V=800.0 PL=0
MOVL C00279 V=800.0 PL=0
MOVL C00280 V=800.0 PL=0
MOVL C00281 V=800.0 PL=0
MOVL C00282 V=800.0 PL=0
MOVL C00283 V=800.0 PL=0
MOVL C00284 V=800.0 PL=0
MOVL C00285 V=800.0 PL=0
MOVL C00286 V=800.0 PL=0
MOVL C00287 V=800.0 PL=0
MOVL C00288 V=800.0 PL=0
MOVL C00289 V=800.0 PL=0
MOVL C00290 V=800.0 PL=0
MOVL C00291 V=800.0 PL=0
MOVL C00292 V=800.0 PL=0
MOVL C00293 V=800.0 PL=0
MOVL C00294 V=800.0 PL=0
MOVL C00295 V=800.0 PL=0
MOVL C00296 V=800.0 PL=0
MOVL C00297 V=800.0 PL=0
MOVL C00298 V=800.0 PL=0
MOVL C00299 V=800.0 PL=0
MOVL C00300 V=800.0 PL=0
MOVL C00301 V=800.0 PL=0
MOVL C00302 V=800.0 PL=0
MOVL C00303 V=800.0 PL=0
MOVL C00304 V=800.0 PL=0
MOVL C00305 V=800.0 PL=0
MOVL C00306 V=800.0 PL=0
MOVL C00307 V=800.0 PL=0
MOVL C00308 V=800.0 PL=0
MOVL C00309 V=800.0 PL=0
MOVL C00310 V=800.0 PL=0
MOVL C00311 V=800.0 PL=0
MOVL C00312 V=800.0 PL=0
MOVL C00313 V=800.0 PL=0
MOVL C00314 V=800.0 PL=0
MOVL C00315 V=800.0 PL=0
MOVL C00316 V=800.0 PL=0
MOVL C00317 V=800.0 PL=0
MOVL C00318 V=800.0 PL=0
MOVL C00319 V=800.0 PL=0
MOVL C00320 V=800.0 PL=0
MOVL C00321 V=800.0 PL=0
MOVL C00322 V=800.0 PL=0
MOVL C00323 V=800.0 PL=0
MOVL C00324 V=800.0 PL=0
MOVL C00325 V=800.0 PL=0
MOVL C00326 V=800.0 PL=0
MOVL C00327 V=800.0 PL=0
MOVL C00328 V=800.0 PL=0
MOVL C00329 V=800.0 PL=0
MOVL C00330 V=800.0 PL=0
MOVL C00331 V=800.0 PL=0
MOVL C00332 V=800.0 PL=0
MOVL C00333 V=800.0 PL=0
MOVL C00334 V=800.0 PL=0
MOVL C00335 V=800.0 PL=0
MOVL C00336 V=800.0 PL=0
MOVL C00337 V=800.0 PL=0
MOVL C00338 V=800.0 PL=0
MOVL C00339 V=800.0 PL=0
MOVL C00340 V=800.0 PL=0
MOVL C00341 V=800.0 PL=0
MOVL C00342 V=800.0 PL=0
MOVL C00343 V=800.0 PL=0
MOVL C00344 V=800.0 PL=0
MOVL C00345 V=800.0 PL=0
MOVL C00346 V=800.0 PL=0
MOVL C00347 V=800.0 PL=0
MOVL C00348 V=800.0 PL=0
MOVL C00349 V=800.0 PL=0
MOVL C00350 V=800.0 PL=0
MOVL C00351 V=800.0 PL=0
MOVL C00352 V=800.0 PL=0
MOVL C00353 V=800.0 PL=0
MOVL C00354 V=800.0 PL=0
MOVL C00355 V=800.0 PL=0
MOVL C00356 V=800.0 PL=0
MOVL C00357 V=800.0 PL=0
MOVL C00358 V=800.0 PL=0
MOVL C00359 V=800.0 PL=0
MOVL C00360 V=800.0 PL=0
MOVL C00361 V=800.0 PL=0
MOVL C00362 V=800.0 PL=0
MOVL C00363 V=800.0 PL=0
MOVL C00364 V=800.0 PL=0
MOVL C00365 V=800.0 PL=0
MOVL C00366 V=800.0 PL=0
MOVL C00367 V=800.0 PL=0
MOVL C00368 V=800.0 PL=0
MOVL C00369 V=800.0 PL=0
MOVL C00370 V=800.0 PL=0
MOVL C00371 V=800.0 PL=0
MOVL C00372 V=800.0 PL=0
MOVL C00373 V=800.0 PL=0
MOVL C00374 V=800.0 PL=0
MOVL C00375 V=800.0 PL=0
MOVL C00376 V=800.0 PL=0
MOVL C00377 V=800.0 PL=0
MOVL C00378 V=800.0 PL=0
MOVL C00379 V=800.0 PL=0
MOVL C00380 V=800.0 PL=0
MOVL C00381 V=800.0 PL=0
MOVL C00382 V=800.0 PL=0
MOVL C00383 V=800.0 PL=0
MOVL C00384 V=800.0 PL=0
MOVL C00385 V=800.0 PL=0
MOVL C00386 V=800.0 PL=0
MOVL C00387 V=800.0 PL=0
MOVL C00388 V=800.0 PL=0
MOVL C00389 V=800.0 PL=0
MOVL C00390 V=800.0 PL=0
MOVL C00391 V=800.0 PL=0
MOVL C00392 V=800.0 PL=0
MOVL C00393 V=800.0 PL=0
MOVL C00394 V=800.0 PL=0
MOVL C00395 V=800.0 PL=0
MOVL C00396 V=800.0 PL=0
MOVL C00397 V=800.0 PL=0
MOVL C00398 V=800.0 PL=0
MOVL C00399 V=800.0 PL=0
MOVL C00400 V=800.0 PL=0
MOVL C00401 V=800.0 PL=0
MOVL C00402 V=800.0 PL=0
MOVL C00403 V=800.0 PL=0
MOVL C00404 V=800.0 PL=0
MOVL C00405 V=800.0 PL=0
MOVL C00406 V=800.0 PL=0
MOVL C00407 V=800.0 PL=0
MOVL C00408 V=800.0 PL=0
MOVL C00409 V=800.0 PL=0
MOVL C00410 V=800.0 PL=0
MOVL C00411 V=800.0 PL=0
MOVL C00412 V=800.0 PL=0
MOVL C00413 V=800.0 PL=0
MOVL C00414 V=800.0 PL=0
MOVL C00415 V=800.0 PL=0
MOVL C00416 V=800.0 PL=0
MOVL C00417 V=800.0 PL=0
MOVL C00418 V=800.0 PL=0
MOVL C00419 V=800.0 PL=0
MOVL C00420 V=800.0 PL=0
MOVL C00421 V=800.0 PL=0
MOVL C00422 V=800.0 PL=0
MOVL C00423 V=800.0 PL=0
MOVL C00424 V=800.0 PL=0
MOVL C00425 V=800.0 PL=0
MOVL C00426 V=800.0 PL=0
MOVL C00427 V=800.0 PL=0
MOVL C00428 V=800.0 PL=0
MOVL C00429 V=800.0 PL=0
MOVL C00430 V=800.0 PL=0
MOVL C00431 V=800.0 PL=0
MOVL C00432 V=800.0 PL=0
MOVL C00433 V=800.0 PL=0
MOVL C00434 V=800.0 PL=0
MOVL C00435 V=800.0 PL=0
MOVL C00436 V=800.0 PL=0
MOVL C00437 V=800.0 PL=0
MOVL C00438 V=800.0 PL=0
MOVL C00439 V=800.0 PL=0
MOVL C00440 V=800.0 PL=0
MOVL C00441 V=800.0 PL=0
MOVL C00442 V=800.0 PL=0
MOVL C00443 V=800.0 PL=0
MOVL C00444 V=800.0 PL=0
MOVL C00445 V=800.0 PL=0
MOVL C00446 V=800.0 PL=0
MOVL C00447 V=800.0 PL=0
MOVL C00448 V=800.0 PL=0
MOVL C00449 V=800.0 PL=0
MOVL C00450 V=800.0 PL=0
MOVL C00451 V=800.0 PL=0
MOVL C00452 V=800.0 PL=0
MOVL C00453 V=800.0 PL=0
MOVL C00454 V=800.0 PL=0
MOVL C00455 V=800.0 PL=0
MOVL C00456 V=800.0 PL=0
MOVL C00457 V=800.0 PL=0
MOVL C00458 V=800.0 PL=0
MOVL C00459 V=800.0 PL=0
MOVL C00460 V=800.0 PL=0
MOVL C00461 V=800.0 PL=0
MOVL C00462 V=800.0 PL=0
MOVL C00463 V=800.0 PL=0
MOVL C00464 V=800.0 PL=0
MOVL C00465 V=800.0 PL=0
MOVL C00466 V=800.0 PL=0
MOVL C00467 V=800.0 PL=0
MOVL C00468 V=800.0 PL=0
MOVL C00469 V=800.0 PL=0
MOVL C00470 V=800.0 PL=0
MOVL C00471 V=800.0 PL=0
MOVL C00472 V=800.0 PL=0
MOVL C00473 V=800.0 PL=0
MOVL C00474 V=800.0 PL=0
MOVL C00475 V=800.0 PL=0
MOVL C00476 V=800.0 PL=0
MOVL C00477 V=800.0 PL=0
MOVL C00478 V=800.0 PL=0
MOVL C00479 V=800.0 PL=0
MOVL C00480 V=800.0 PL=0
MOVL C00481 V=800.0 PL=0
MOVL C00482 V=800.0 PL=0
MOVL C00483 V=800.0 PL=0
MOVL C00484 V=800.0 PL=0
MOVL C00485 V=800.0 PL=0
MOVL C00486 V=800.0 PL=0
MOVL C00487 V=800.0 PL=0
MOVL C00488 V=800.0 PL=0
MOVL C00489 V=800.0 PL=0
MOVL C00490 V=800.0 PL=0
MOVL C00491 V=800.0 PL=0
MOVL C00492 V=800.0 PL=0
MOVL C00493 V=800.0 PL=0
MOVL C00494 V=800.0 PL=0
MOVL C00495 V=800.0 PL=0
MOVL C00496 V=800.0 PL=0
MOVL C00497 V=800.0 PL=0
MOVL C00498 V=800.0 PL=0
MOVL C00499 V=800.0 PL=0
MOVL C00500 V=800.0 PL=0
MOVL C00501 V=800.0 PL=0
MOVL C00502 V=800.0 PL=0
MOVL C00503 V=800.0 PL=0
MOVL C00504 V=800.0 PL=0
MOVL C00505 V=800.0 PL=0
MOVL C00506 V=800.0 PL=0
MOVL C00507 V=800.0 PL=0
MOVL C00508 V=800.0 PL=0
MOVL C00509 V=800.0 PL=0
MOVL C00510 V=800.0 PL=0
MOVL C00511 V=800.0 PL=0
MOVL C00512 V=800.0 PL=0
MOVL C00513 V=800.0 PL=0
MOVL C00514 V=800.0 PL=0
MOVL C00515 V=800.0 PL=0
MOVL C00516 V=800.0 PL=0
MOVL C00517 V=800.0 PL=0
MOVL C00518 V=800.0 PL=0
MOVL C00519 V=800.0 PL=0
MOVL C00520 V=800.0 PL=0
MOVL C00521 V=800.0 PL=0
MOVL C00522 V=800.0 PL=0
MOVL C00523 V=800.0 PL=0
MOVL C00524 V=800.0 PL=0
MOVL C00525 V=800.0 PL=0
MOVL C00526 V=800.0 PL=0
MOVL C00527 V=800.0 PL=0
MOVL C00528 V=800.0 PL=0
MOVL C00529 V=800.0 PL=0
MOVL C00530 V=800.0 PL=0
MOVL C00531 V=800.0 PL=0
MOVL C00532 V=800.0 PL=0
MOVL C00533 V=800.0 PL=0
MOVL C00534 V=800.0 PL=0
MOVL C00535 V=800.0 PL=0
MOVL C00536 V=800.0 PL=0
MOVL C00537 V=800.0 PL=0
MOVL C00538 V=800.0 PL=0
MOVL C00539 V=800.0 PL=0
MOVL C00540 V=800.0 PL=0
MOVL C00541 V=800.0 PL=0
MOVL C00542 V=800.0 PL=0
MOVL C00543 V=800.0 PL=0
MOVL C00544 V=800.0 PL=0
MOVL C00545 V=800.0 PL=0
MOVL C00546 V=800.0 PL=0
MOVL C00547 V=800.0 PL=0
MOVL C00548 V=800.0 PL=0
MOVL C00549 V=800.0 PL=0
MOVL C00550 V=800.0 PL=0
MOVL C00551 V=800.0 PL=0
MOVL C00552 V=800.0 PL=0
MOVL C00553 V=800.0 PL=0
MOVL C00554 V=800.0 PL=0
MOVL C00555 V=800.0 PL=0
MOVL C00556 V=800.0 PL=0
MOVL C00557 V=800.0 PL=0
MOVL C00558 V=800.0 PL=0
MOVL C00559 V=800.0 PL=0
MOVL C00560 V=800.0 PL=0
MOVL C00561 V=800.0 PL=0
MOVL C00562 V=800.0 PL=0
MOVL C00563 V=800.0 PL=0
MOVL C00564 V=800.0 PL=0
MOVL C00565 V=800.0 PL=0
MOVL C00566 V=800.0 PL=0
MOVL C00567 V=800.0 PL=0
MOVL C00568 V=800.0 PL=0
MOVL C00569 V=800.0 PL=0
MOVL C00570 V=800.0 PL=0
MOVL C00571 V=800.0 PL=0
MOVL C00572 V=800.0 PL=0
MOVL C00573 V=800.0 PL=0
MOVL C00574 V=800.0 PL=0
MOVL C00575 V=800.0 PL=0
MOVL C00576 V=800.0 PL=0
MOVL C00577 V=800.0 PL=0
MOVL C00578 V=800.0 PL=0
MOVL C00579 V=800.0 PL=0
MOVL C00580 V=800.0 PL=0
MOVL C00581 V=800.0 PL=0
MOVL C00582 V=800.0 PL=0
MOVL C00583 V=800.0 PL=0
MOVL C00584 V=800.0 PL=0
MOVL C00585 V=800.0 PL=0
MOVL C00586 V=800.0 PL=0
MOVL C00587 V=800.0 PL=0
MOVL C00588 V=800.0 PL=0
MOVL C00589 V=800.0 PL=0
MOVL C00590 V=800.0 PL=0
MOVL C00591 V=800.0 PL=0
MOVL C00592 V=800.0 PL=0
MOVL C00593 V=800.0 PL=0
MOVL C00594 V=800.0 PL=0
MOVL C00595 V=800.0 PL=0
MOVL C00596 V=800.0 PL=0
MOVL C00597 V=800.0 PL=0
MOVL C00598 V=800.0 PL=0
MOVL C00599 V=800.0 PL=0
MOVL C00600 V=800.0 PL=0
MOVL C00601 V=800.0 PL=0
MOVL C00602 V=800.0 PL=0
MOVL C00603 V=800.0 PL=0
MOVL C00604 V=800.0 PL=0
MOVL C00605 V=800.0 PL=0
MOVL C00606 V=800.0 PL=0
MOVL C00607 V=800.0 PL=0
MOVL C00608 V=800.0 PL=0
MOVL C00609 V=800.0 PL=0
MOVL C00610 V=800.0 PL=0
MOVL C00611 V=800.0 PL=0
MOVL C00612 V=800.0 PL=0
MOVL C00613 V=800.0 PL=0
MOVL C00614 V=800.0 PL=0
MOVL C00615 V=800.0 PL=0
MOVL C00616 V=800.0 PL=0
MOVL C00617 V=800.0 PL=0
MOVL C00618 V=800.0 PL=0
MOVL C00619 V=800.0 PL=0
MOVL C00620 V=800.0 PL=0
MOVL C00621 V=800.0 PL=0
MOVL C00622 V=800.0 PL=0
MOVL C00623 V=800.0 PL=0
MOVL C00624 V=800.0 PL=0
MOVL C00625 V=800.0 PL=0
MOVL C00626 V=800.0 PL=0
MOVL C00627 V=800.0 PL=0
MOVL C00628 V=800.0 PL=0
MOVL C00629 V=800.0 PL=0
MOVL C00630 V=800.0 PL=0
MOVL C00631 V=800.0 PL=0
MOVL C00632 V=800.0 PL=0
MOVL C00633 V=800.0 PL=0
MOVL C00634 V=800.0 PL=0
MOVL C00635 V=800.0 PL=0
MOVL C00636 V=800.0 PL=0
MOVL C00637 V=800.0 PL=0
MOVL C00638 V=800.0 PL=0
MOVL C00639 V=800.0 PL=0
MOVL C00640 V=800.0 PL=0
MOVL C00641 V=800.0 PL=0
MOVL C00642 V=800.0 PL=0
MOVL C00643 V=800.0 PL=0
MOVL C00644 V=800.0 PL=0
MOVL C00645 V=800.0 PL=0
MOVL C00646 V=800.0 PL=0
MOVL C00647 V=800.0 PL=0
MOVL C00648 V=800.0 PL=0
MOVL C00649 V=800.0 PL=0
MOVL C00650 V=800.0 PL=0
MOVL C00651 V=800.0 PL=0
MOVL C00652 V=800.0 PL=0
MOVL C00653 V=800.0 PL=0
MOVL C00654 V=800.0 PL=0
MOVL C00655 V=800.0 PL=0
MOVL C00656 V=800.0 PL=0
MOVL C00657 V=800.0 PL=0
MOVL C00658 V=800.0 PL=0
MOVL C00659 V=800.0 PL=0
MOVL C00660 V=800.0 PL=0
MOVL C00661 V=800.0 PL=0
MOVL C00662 V=800.0 PL=0
MOVL C00663 V=800.0 PL=0
MOVL C00664 V=800.0 PL=0
MOVL C00665 V=800.0 PL=0
MOVL C00666 V=800.0 PL=0
MOVL C00667 V=800.0 PL=0
MOVL C00668 V=800.0 PL=0
MOVL C00669 V=800.0 PL=0
MOVL C00670 V=800.0 PL=0
MOVL C00671 V=800.0 PL=0
MOVL C00672 V=800.0 PL=0
MOVL C00673 V=800.0 PL=0
MOVL C00674 V=800.0 PL=0
MOVL C00675 V=800.0 PL=0
MOVL C00676 V=800.0 PL=0
MOVL C00677 V=800.0 PL=0
MOVL C00678 V=800.0 PL=0
MOVL C00679 V=800.0 PL=0
MOVL C00680 V=800.0 PL=0
MOVL C00681 V=800.0 PL=0
MOVL C00682 V=800.0 PL=0
MOVL C00683 V=800.0 PL=0
MOVL C00684 V=800.0 PL=0
MOVL C00685 V=800.0 PL=0
MOVL C00686 V=800.0 PL=0
MOVL C00687 V=800.0 PL=0
MOVL C00688 V=800.0 PL=0
MOVL C00689 V=800.0 PL=0
MOVL C00690 V=800.0 PL=0
MOVL C00691 V=800.0 PL=0
MOVL C00692 V=800.0 PL=0
MOVL C00693 V=800.0 PL=0
MOVL C00694 V=800.0 PL=0
MOVL C00695 V=800.0 PL=0
MOVL C00696 V=800.0 PL=0
MOVL C00697 V=800.0 PL=0
MOVL C00698 V=800.0 PL=0
MOVL C00699 V=800.0 PL=0
MOVL C00700 V=800.0 PL=0
MOVL C00701 V=800.0 PL=0
MOVL C00702 V=800.0 PL=0
MOVL C00703 V=800.0 PL=0
MOVL C00704 V=800.0 PL=0
MOVL C00705 V=800.0 PL=0
MOVL C00706 V=800.0 PL=0
MOVL C00707 V=800.0 PL=0
MOVL C00708 V=800.0 PL=0
MOVL C00709 V=800.0 PL=0
MOVL C00710 V=800.0 PL=0
MOVL C00711 V=800.0 PL=0
MOVL C00712 V=800.0 PL=0
MOVL C00713 V=800.0 PL=0
MOVL C00714 V=800.0 PL=0
MOVL C00715 V=800.0 PL=0
MOVL C00716 V=800.0 PL=0
MOVL C00717 V=800.0 PL=0
MOVL C00718 V=800.0 PL=0
MOVL C00719 V=800.0 PL=0
MOVL C00720 V=800.0 PL=0
MOVL C00721 V=800.0 PL=0
MOVL C00722 V=800.0 PL=0
MOVL C00723 V=800.0 PL=0
MOVL C00724 V=800.0 PL=0
MOVL C00725 V=800.0 PL=0
MOVL C00726 V=800.0 PL=0
MOVL C00727 V=800.0 PL=0
MOVL C00728 V=800.0 PL=0
MOVL C00729 V=800.0 PL=0
MOVL C00730 V=800.0 PL=0
MOVL C00731 V=800.0 PL=0
MOVL C00732 V=800.0 PL=0
MOVL C00733 V=800.0 PL=0
MOVL C00734 V=800.0 PL=0
MOVL C00735 V=800.0 PL=0
MOVL C00736 V=800.0 PL=0
MOVL C00737 V=800.0 PL=0
MOVL C00738 V=800.0 PL=0
MOVL C00739 V=800.0 PL=0
MOVL C00740 V=800.0 PL=0
MOVL C00741 V=800.0 PL=0
MOVL C00742 V=800.0 PL=0
MOVL C00743 V=800.0 PL=0
MOVL C00744 V=800.0 PL=0
MOVL C00745 V=800.0 PL=0
MOVL C00746 V=800.0 PL=0
MOVL C00747 V=800.0 PL=0
MOVL C00748 V=800.0 PL=0
MOVL C00749 V=800.0 PL=0
MOVL C00750 V=800.0 PL=0
MOVL C00751 V=800.0 PL=0
MOVL C00752 V=800.0 PL=0
MOVL C00753 V=800.0 PL=0
MOVL C00754 V=800.0 PL=0
MOVL C00755 V=800.0 PL=0
MOVL C00756 V=800.0 PL=0
MOVL C00757 V=800.0 PL=0
MOVL C00758 V=800.0 PL=0
MOVL C00759 V=800.0 PL=0
MOVL C00760 V=800.0 PL=0
MOVL C00761 V=800.0 PL=0
MOVL C00762 V=800.0 PL=0
MOVL C00763 V=800.0 PL=0
MOVL C00764 V=800.0 PL=0
MOVL C00765 V=800.0 PL=0
MOVL C00766 V=800.0 PL=0
MOVL C00767 V=800.0 PL=0
MOVL C00768 V=800.0 PL=0
MOVL C00769 V=800.0 PL=0
MOVL C00770 V=800.0 PL=0
MOVL C00771 V=800.0 PL=0
MOVL C00772 V=800.0 PL=0
MOVL C00773 V=800.0 PL=0
MOVL C00774 V=800.0 PL=0
MOVL C00775 V=800.0 PL=0
MOVL C00776 V=800.0 PL=0
MOVL C00777 V=800.0 PL=0
MOVL C00778 V=800.0 PL=0
MOVL C00779 V=800.0 PL=0
MOVL C00780 V=800.0 PL=0
MOVL C00781 V=800.0 PL=0
MOVL C00782 V=800.0 PL=0
MOVL C00783 V=800.0 PL=0
MOVL C00784 V=800.0 PL=0
MOVL C00785 V=800.0 PL=0
MOVL C00786 V=800.0 PL=0
MOVL C00787 V=800.0 PL=0
MOVL C00788 V=800.0 PL=0
MOVL C00789 V=800.0 PL=0
MOVL C00790 V=800.0 PL=0
MOVL C00791 V=800.0 PL=0
MOVL C00792 V=800.0 PL=0
MOVL C00793 V=800.0 PL=0
MOVL C00794 V=800.0 PL=0
MOVL C00795 V=800.0 PL=0
MOVL C00796 V=800.0 PL=0
MOVL C00797 V=800.0 PL=0
MOVL C00798 V=800.0 PL=0
MOVL C00799 V=800.0 PL=0
MOVL C00800 V=800.0 PL=0
MOVL C00801 V=800.0 PL=0
MOVL C00802 V=800.0 PL=0
MOVL C00803 V=800.0 PL=0
MOVL C00804 V=800.0 PL=0
MOVL C00805 V=800.0 PL=0
MOVL C00806 V=800.0 PL=0
MOVL C00807 V=800.0 PL=0
MOVL C00808 V=800.0 PL=0
MOVL C00809 V=800.0 PL=0
MOVL C00810 V=800.0 PL=0
MOVL C00811 V=800.0 PL=0
MOVL C00812 V=800.0 PL=0
MOVL C00813 V=800.0 PL=0
MOVL C00814 V=800.0 PL=0
MOVL C00815 V=800.0 PL=0
MOVL C00816 V=800.0 PL=0
MOVL C00817 V=800.0 PL=0
MOVL C00818 V=800.0 PL=0
MOVL C00819 V=800.0 PL=0
MOVL C00820 V=800.0 PL=0
MOVL C00821 V=800.0 PL=0
MOVL C00822 V=800.0 PL=0
MOVL C00823 V=800.0 PL=0
MOVL C00824 V=800.0 PL=0
MOVL C00825 V=800.0 PL=0
MOVL C00826 V=800.0 PL=0
MOVL C00827 V=800.0 PL=0
MOVL C00828 V=800.0 PL=0
MOVL C00829 V=800.0 PL=0
MOVL C00830 V=800.0 PL=0
MOVL C00831 V=800.0 PL=0
MOVL C00832 V=800.0 PL=0
MOVL C00833 V=800.0 PL=0
MOVL C00834 V=800.0 PL=0
MOVL C00835 V=800.0 PL=0
MOVL C00836 V=800.0 PL=0
MOVL C00837 V=800.0 PL=0
MOVL C00838 V=800.0 PL=0
MOVL C00839 V=800.0 PL=0
MOVL C00840 V=800.0 PL=0
MOVL C00841 V=800.0 PL=0
MOVL C00842 V=800.0 PL=0
MOVL C00843 V=800.0 PL=0
MOVL C00844 V=800.0 PL=0
MOVL C00845 V=800.0 PL=0
MOVL C00846 V=800.0 PL=0
MOVL C00847 V=800.0 PL=0
MOVL C00848 V=800.0 PL=0
MOVL C00849 V=800.0 PL=0
MOVL C00850 V=800.0 PL=0
MOVL C00851 V=800.0 PL=0
MOVL C00852 V=800.0 PL=0
MOVL C00853 V=800.0 PL=0
MOVL C00854 V=800.0 PL=0
MOVL C00855 V=800.0 PL=0
MOVL C00856 V=800.0 PL=0
MOVL C00857 V=800.0 PL=0
MOVL C00858 V=800.0 PL=0
MOVL C00859 V=800.0 PL=0
MOVL C00860 V=800.0 PL=0
MOVL C00861 V=800.0 PL=0
MOVL C00862 V=800.0 PL=0
MOVL C00863 V=800.0 PL=0
MOVL C00864 V=800.0 PL=0
MOVL C00865 V=800.0 PL=0
MOVL C00866 V=800.0 PL=0
MOVL C00867 V=800.0 PL=0
MOVL C00868 V=800.0 PL=0
MOVL C00869 V=800.0 PL=0
MOVL C00870 V=800.0 PL=0
MOVL C00871 V=800.0 PL=0
MOVL C00872 V=800.0 PL=0
MOVL C00873 V=800.0 PL=0
MOVL C00874 V=800.0 PL=0
MOVL C00875 V=800.0 PL=0
MOVL C00876 V=800.0 PL=0
MOVL C00877 V=800.0 PL=0
MOVL C00878 V=800.0 PL=0
MOVL C00879 V=800.0 PL=0
MOVL C00880 V=800.0 PL=0
MOVL C00881 V=800.0 PL=0
MOVL C00882 V=800.0 PL=0
MOVL C00883 V=800.0 PL=0
MOVL C00884 V=800.0 PL=0
MOVL C00885 V=800.0 PL=0
MOVL C00886 V=800.0 PL=0
MOVL C00887 V=800.0 PL=0
MOVL C00888 V=800.0 PL=0
MOVL C00889 V=800.0 PL=0
MOVL C00890 V=800.0 PL=0
MOVL C00891 V=800.0 PL=0
MOVL C00892 V=800.0 PL=0
MOVL C00893 V=800.0 PL=0
MOVL C00894 V=800.0 PL=0
MOVL C00895 V=800.0 PL=0
MOVL C00896 V=800.0 PL=0
MOVL C00897 V=800.0 PL=0
MOVL C00898 V=800.0 PL=0
MOVL C00899 V=800.0 PL=0
MOVL C00900 V=800.0 PL=0
MOVL C00901 V=800.0 PL=0
MOVL C00902 V=800.0 PL=0
MOVL C00903 V=800.0 PL=0
MOVL C00904 V=800.0 PL=0
MOVL C00905 V=800.0 PL=0
MOVL C00906 V=800.0 PL=0
MOVL C00907 V=800.0 PL=0
MOVL C00908 V=800.0 PL=0
MOVL C00909 V=800.0 PL=0
MOVL C00910 V=800.0 PL=0
MOVL C00911 V=800.0 PL=0
MOVL C00912 V=800.0 PL=0
MOVL C00913 V=800.0 PL=0
MOVL C00914 V=800.0 PL=0
MOVL C00915 V=800.0 PL=0
MOVL C00916 V=800.0 PL=0
MOVL C00917 V=800.0 PL=0
MOVL C00918 V=800.0 PL=0
MOVL C00919 V=800.0 PL=0
MOVL C00920 V=800.0 PL=0
MOVL C00921 V=800.0 PL=0
MOVL C00922 V=800.0 PL=0
MOVL C00923 V=800.0 PL=0
MOVL C00924 V=800.0 PL=0
MOVL C00925 V=800.0 PL=0
MOVL C00926 V=800.0 PL=0
MOVL C00927 V=800.0 PL=0
MOVL C00928 V=800.0 PL=0
MOVL C00929 V=800.0 PL=0
MOVL C00930 V=800.0 PL=0
MOVL C00931 V=800.0 PL=0
MOVL C00932 V=800.0 PL=0
MOVL C00933 V=800.0 PL=0
MOVL C00934 V=800.0 PL=0
MOVL C00935 V=800.0 PL=0
MOVL C00936 V=800.0 PL=0
MOVL C00937 V=800.0 PL=0
MOVL C00938 V=800.0 PL=0
MOVL C00939 V=800.0 PL=0
MOVL C00940 V=800.0 PL=0
MOVL C00941 V=800.0 PL=0
MOVL C00942 V=800.0 PL=0
MOVL C00943 V=800.0 PL=0
MOVL C00944 V=800.0 PL=0
MOVL C00945 V=800.0 PL=0
MOVL C00946 V=800.0 PL=0
MOVL C00947 V=800.0 PL=0
MOVL C00948 V=800.0 PL=0
MOVL C00949 V=800.0 PL=0
MOVL C00950 V=800.0 PL=0
MOVL C00951 V=800.0 PL=0
MOVL C00952 V=800.0 PL=0
MOVL C00953 V=800.0 PL=0
MOVL C00954 V=800.0 PL=0
MOVL C00955 V=800.0 PL=0
MOVL C00956 V=800.0 PL=0
MOVL C00957 V=800.0 PL=0
MOVL C00958 V=800.0 PL=0
MOVL C00959 V=800.0 PL=0
MOVL C00960 V=800.0 PL=0
MOVL C00961 V=800.0 PL=0
MOVL C00962 V=800.0 PL=0
MOVL C00963 V=800.0 PL=0
MOVL C00964 V=800.0 PL=0
MOVL C00965 V=800.0 PL=0
MOVL C00966 V=800.0 PL=0
MOVL C00967 V=800.0 PL=0
MOVL C00968 V=800.0 PL=0
MOVL C00969 V=800.0 PL=0
MOVL C00970 V=800.0 PL=0
MOVL C00971 V=800.0 PL=0
MOVL C00972 V=800.0 PL=0
MOVL C00973 V=800.0 PL=0
MOVL C00974 V=800.0 PL=0
MOVL C00975 V=800.0 PL=0
MOVL C00976 V=800.0 PL=0
MOVL C00977 V=800.0 PL=0
MOVL C00978 V=800.0 PL=0
MOVL C00979 V=800.0 PL=0
MOVL C00980 V=800.0 PL=0
MOVL C00981 V=800.0 PL=0
MOVL C00982 V=800.0 PL=0
MOVL C00983 V=800.0 PL=0
MOVL C00984 V=800.0 PL=0
MOVL C00985 V=800.0 PL=0
MOVL C00986 V=800.0 PL=0
MOVL C00987 V=800.0 PL=0
MOVL C00988 V=800.0 PL=0
MOVL C00989 V=800.0 PL=0
MOVL C00990 V=800.0 PL=0
MOVL C00991 V=800.0 PL=0
MOVL C00992 V=800.0 PL=0
MOVL C00993 V=800.0 PL=0
MOVL C00994 V=800.0 PL=0
MOVL C00995 V=800.0 PL=0
MOVL C00996 V=800.0 PL=0
MOVL C00997 V=800.0 PL=0
MOVL C00998 V=800.0 PL=0
MOVL C00999 V=800.0 PL=0
MOVL C01000 V=800.0 PL=0
MOVL C01001 V=800.0 PL=0
MOVL C01002 V=800.0 PL=0
MOVL C01003 V=800.0 PL=0
MOVL C01004 V=800.0 PL=0
MOVL C01005 V=800.0 PL=0
MOVL C01006 V=800.0 PL=0
MOVL C01007 V=800.0 PL=0
MOVL C01008 V=800.0 PL=0
MOVL C01009 V=800.0 PL=0
MOVL C01010 V=800.0 PL=0
MOVL C01011 V=800.0 PL=0
MOVL C01012 V=800.0 PL=0
MOVL C01013 V=800.0 PL=0
MOVL C01014 V=800.0 PL=0
MOVL C01015 V=800.0 PL=0
MOVL C01016 V=800.0 PL=0
MOVL C01017 V=800.0 PL=0
MOVL C01018 V=800.0 PL=0
MOVL C01019 V=800.0 PL=0
MOVL C01020 V=800.0 PL=0
MOVL C01021 V=800.0 PL=0
MOVL C01022 V=800.0 PL=0
MOVL C01023 V=800.0 PL=0
MOVL C01024 V=800.0 PL=0
MOVL C01025 V=800.0 PL=0
MOVL C01026 V=800.0 PL=0
MOVL C01027 V=800.0 PL=0
MOVL C01028 V=800.0 PL=0
MOVL C01029 V=800.0 PL=0
MOVL C01030 V=800.0 PL=0
MOVL C01031 V=800.0 PL=0
MOVL C01032 V=800.0 PL=0
MOVL C01033 V=800.0 PL=0
MOVL C01034 V=800.0 PL=0
MOVL C01035 V=800.0 PL=0
MOVL C01036 V=800.0 PL=0
MOVL C01037 V=800.0 PL=0
MOVL C01038 V=800.0 PL=0
MOVL C01039 V=800.0 PL=0
MOVL C01040 V=800.0 PL=0
MOVL C01041 V=800.0 PL=0
MOVL C01042 V=800.0 PL=0
MOVL C01043 V=800.0 PL=0
MOVL C01044 V=800.0 PL=0
MOVL C01045 V=800.0 PL=0
MOVL C01046 V=800.0 PL=0
MOVL C01047 V=800.0 PL=0
MOVL C01048 V=800.0 PL=0
MOVL C01049 V=800.0 PL=0
MOVL C01050 V=800.0 PL=0
MOVL C01051 V=800.0 PL=0
MOVL C01052 V=800.0 PL=0
MOVL C01053 V=800.0 PL=0
MOVL C01054 V=800.0 PL=0
MOVL C01055 V=800.0 PL=0
MOVL C01056 V=800.0 PL=0
MOVL C01057 V=800.0 PL=0
MOVL C01058 V=800.0 PL=0
MOVL C01059 V=800.0 PL=0
MOVL C01060 V=800.0 PL=0
MOVL C01061 V=800.0 PL=0
MOVL C01062 V=800.0 PL=0
MOVL C01063 V=800.0 PL=0
MOVL C01064 V=800.0 PL=0
MOVL C01065 V=800.0 PL=0
MOVL C01066 V=800.0 PL=0
MOVL C01067 V=800.0 PL=0
MOVL C01068 V=800.0 PL=0
MOVL C01069 V=800.0 PL=0
MOVL C01070 V=800.0 PL=0
MOVL C01071 V=800.0 PL=0
MOVL C01072 V=800.0 PL=0
MOVL C01073 V=800.0 PL=0
MOVL C01074 V=800.0 PL=0
MOVL C01075 V=800.0 PL=0
MOVL C01076 V=800.0 PL=0
MOVL C01077 V=800.0 PL=0
MOVL C01078 V=800.0 PL=0
MOVL C01079 V=800.0 PL=0
MOVL C01080 V=800.0 PL=0
MOVL C01081 V=800.0 PL=0
MOVL C01082 V=800.0 PL=0
MOVL C01083 V=800.0 PL=0
MOVL C01084 V=800.0 PL=0
MOVL C01085 V=800.0 PL=0
MOVL C01086 V=800.0 PL=0
MOVL C01087 V=800.0 PL=0
MOVL C01088 V=800.0 PL=0
MOVL C01089 V=800.0 PL=0
MOVL C01090 V=800.0 PL=0
MOVL C01091 V=800.0 PL=0
MOVL C01092 V=800.0 PL=0
MOVL C01093 V=800.0 PL=0
MOVL C01094 V=800.0 PL=0
MOVL C01095 V=800.0 PL=0
MOVL C01096 V=800.0 PL=0
MOVL C01097 V=800.0 PL=0
MOVL C01098 V=800.0 PL=0
MOVL C01099 V=800.0 PL=0
MOVL C01100 V=800.0 PL=0
MOVL C01101 V=800.0 PL=0
MOVL C01102 V=800.0 PL=0
MOVL C01103 V=800.0 PL=0
MOVL C01104 V=800.0 PL=0
MOVL C01105 V=800.0 PL=0
MOVL C01106 V=800.0 PL=0
MOVL C01107 V=800.0 PL=0
MOVL C01108 V=800.0 PL=0
MOVL C01109 V=800.0 PL=0
MOVL C01110 V=800.0 PL=0
MOVL C01111 V=800.0 PL=0
MOVL C01112 V=800.0 PL=0
MOVL C01113 V=800.0 PL=0
MOVL C01114 V=800.0 PL=0
MOVL C01115 V=800.0 PL=0
MOVL C01116 V=800.0 PL=0
MOVL C01117 V=800.0 PL=0
MOVL C01118 V=800.0 PL=0
MOVL C01119 V=800.0 PL=0
MOVL C01120 V=800.0 PL=0
MOVL C01121 V=800.0 PL=0
MOVL C01122 V=800.0 PL=0
MOVL C01123 V=800.0 PL=0
MOVL C01124 V=800.0 PL=0
MOVL C01125 V=800.0 PL=0
MOVL C01126 V=800.0 PL=0
MOVL C01127 V=800.0 PL=0
MOVL C01128 V=800.0 PL=0
MOVL C01129 V=800.0 PL=0
MOVL C01130 V=800.0 PL=0
MOVL C01131 V=800.0 PL=0
MOVL C01132 V=800.0 PL=0
MOVL C01133 V=800.0 PL=0
MOVL C01134 V=800.0 PL=0
MOVL C01135 V=800.0 PL=0
MOVL C01136 V=800.0 PL=0
MOVL C01137 V=800.0 PL=0
MOVL C01138 V=800.0 PL=0
MOVL C01139 V=800.0 PL=0
MOVL C01140 V=800.0 PL=0
MOVL C01141 V=800.0 PL=0
MOVL C01142 V=800.0 PL=0
MOVL C01143 V=800.0 PL=0
MOVL C01144 V=800.0 PL=0
MOVL C01145 V=800.0 PL=0
MOVL C01146 V=800.0 PL=0
MOVL C01147 V=800.0 PL=0
MOVL C01148 V=800.0 PL=0
MOVL C01149 V=800.0 PL=0
MOVL C01150 V=800.0 PL=0
MOVL C01151 V=800.0 PL=0
MOVL C01152 V=800.0 PL=0
MOVL C01153 V=800.0 PL=0
MOVL C01154 V=800.0 PL=0
MOVL C01155 V=800.0 PL=0
MOVL C01156 V=800.0 PL=0
MOVL C01157 V=800.0 PL=0
MOVL C01158 V=800.0 PL=0
MOVL C01159 V=800.0 PL=0
MOVL C01160 V=800.0 PL=0
MOVL C01161 V=800.0 PL=0
MOVL C01162 V=800.0 PL=0
MOVL C01163 V=800.0 PL=0
MOVL C01164 V=800.0 PL=0
MOVL C01165 V=800.0 PL=0
MOVL C01166 V=800.0 PL=0
MOVL C01167 V=800.0 PL=0
MOVL C01168 V=800.0 PL=0
MOVL C01169 V=800.0 PL=0
MOVL C01170 V=800.0 PL=0
MOVL C01171 V=800.0 PL=0
MOVL C01172 V=800.0 PL=0
MOVL C01173 V=800.0 PL=0
MOVL C01174 V=800.0 PL=0
MOVL C01175 V=800.0 PL=0
MOVL C01176 V=800.0 PL=0
MOVL C01177 V=800.0 PL=0
MOVL C01178 V=800.0 PL=0
MOVL C01179 V=800.0 PL=0
MOVL C01180 V=800.0 PL=0
MOVL C01181 V=800.0 PL=0
MOVL C01182 V=800.0 PL=0
MOVL C01183 V=800.0 PL=0
MOVL C01184 V=800.0 PL=0
MOVL C01185 V=800.0 PL=0
MOVL C01186 V=800.0 PL=0
MOVL C01187 V=800.0 PL=0
MOVL C01188 V=800.0 PL=0
MOVL C01189 V=800.0 PL=0
MOVL C01190 V=800.0 PL=0
MOVL C01191 V=800.0 PL=0
MOVL C01192 V=800.0 PL=0
MOVL C01193 V=800.0 PL=0
MOVL C01194 V=800.0 PL=0
MOVL C01195 V=800.0 PL=0
MOVL C01196 V=800.0 PL=0
MOVL C01197 V=800.0 PL=0
MOVL C01198 V=800.0 PL=0
MOVL C01199 V=800.0 PL=0
MOVL C01200 V=800.0 PL=0
MOVL C01201 V=800.0 PL=0
MOVL C01202 V=800.0 PL=0
MOVL C01203 V=800.0 PL=0
MOVL C01204 V=800.0 PL=0
MOVL C01205 V=800.0 PL=0
MOVL C01206 V=800.0 PL=0
MOVL C01207 V=800.0 PL=0
MOVL C01208 V=800.0 PL=0
MOVL C01209 V=800.0 PL=0
MOVL C01210 V=800.0 PL=0
MOVL C01211 V=800.0 PL=0
MOVL C01212 V=800.0 PL=0
MOVL C01213 V=800.0 PL=0
MOVL C01214 V=800.0 PL=0
MOVL C01215 V=800.0 PL=0
MOVL C01216 V=800.0 PL=0
MOVL C01217 V=800.0 PL=0
MOVL C01218 V=800.0 PL=0
MOVL C01219 V=800.0 PL=0
MOVL C01220 V=800.0 PL=0
MOVL C01221 V=800.0 PL=0
MOVL C01222 V=800.0 PL=0
MOVL C01223 V=800.0 PL=0
MOVL C01224 V=800.0 PL=0
MOVL C01225 V=800.0 PL=0
MOVL C01226 V=800.0 PL=0
MOVL C01227 V=800.0 PL=0
MOVL C01228 V=800.0 PL=0
MOVL C01229 V=800.0 PL=0
MOVL C01230 V=800.0 PL=0
MOVL C01231 V=800.0 PL=0
MOVL C01232 V=800.0 PL=0
MOVL C01233 V=800.0 PL=0
MOVL C01234 V=800.0 PL=0
MOVL C01235 V=800.0 PL=0
MOVL C01236 V=800.0 PL=0
MOVL C01237 V=800.0 PL=0
MOVL C01238 V=800.0 PL=0
MOVL C01239 V=800.0 PL=0
MOVL C01240 V=800.0 PL=0
MOVL C01241 V=800.0 PL=0
MOVL C01242 V=800.0 PL=0
MOVL C01243 V=800.0 PL=0
MOVL C01244 V=800.0 PL=0
MOVL C01245 V=800.0 PL=0
MOVL C01246 V=800.0 PL=0
MOVL C01247 V=800.0 PL=0
MOVL C01248 V=800.0 PL=0
MOVL C01249 V=800.0 PL=0
MOVL C01250 V=800.0 PL=0
MOVL C01251 V=800.0 PL=0
MOVL C01252 V=800.0 PL=0
MOVL C01253 V=800.0 PL=0
MOVL C01254 V=800.0 PL=0
MOVL C01255 V=800.0 PL=0
MOVL C01256 V=800.0 PL=0
MOVL C01257 V=800.0 PL=0
MOVL C01258 V=800.0 PL=0
MOVL C01259 V=800.0 PL=0
MOVL C01260 V=800.0 PL=0
MOVL C01261 V=800.0 PL=0
MOVL C01262 V=800.0 PL=0
MOVL C01263 V=800.0 PL=0
MOVL C01264 V=800.0 PL=0
MOVL C01265 V=800.0 PL=0
MOVL C01266 V=800.0 PL=0
MOVL C01267 V=800.0 PL=0
MOVL C01268 V=800.0 PL=0
MOVL C01269 V=800.0 PL=0
MOVL C01270 V=800.0 PL=0
MOVL C01271 V=800.0 PL=0
MOVL C01272 V=800.0 PL=0
MOVL C01273 V=800.0 PL=0
MOVL C01274 V=800.0 PL=0
MOVL C01275 V=800.0 PL=0
MOVL C01276 V=800.0 PL=0
MOVL C01277 V=800.0 PL=0
MOVL C01278 V=800.0 PL=0
MOVL C01279 V=800.0 PL=0
MOVL C01280 V=800.0 PL=0
MOVL C01281 V=800.0 PL=0
MOVL C01282 V=800.0 PL=0
MOVL C01283 V=800.0 PL=0
MOVL C01284 V=800.0 PL=0
MOVL C01285 V=800.0 PL=0
MOVL C01286 V=800.0 PL=0
MOVL C01287 V=800.0 PL=0
MOVL C01288 V=800.0 PL=0
MOVL C01289 V=800.0 PL=0
MOVL C01290 V=800.0 PL=0
MOVL C01291 V=800.0 PL=0
MOVL C01292 V=800.0 PL=0
MOVL C01293 V=800.0 PL=0
MOVL C01294 V=800.0 PL=0
MOVL C01295 V=800.0 PL=0
MOVL C01296 V=800.0 PL=0
MOVL C01297 V=800.0 PL=0
MOVL C01298 V=800.0 PL=0
MOVL C01299 V=800.0 PL=0
MOVL C01300 V=800.0 PL=0
MOVL C01301 V=800.0 PL=0
MOVL C01302 V=800.0 PL=0
MOVL C01303 V=800.0 PL=0
MOVL C01304 V=800.0 PL=0
MOVL C01305 V=800.0 PL=0
MOVL C01306 V=800.0 PL=0
MOVL C01307 V=800.0 PL=0
MOVL C01308 V=800.0 PL=0
MOVL C01309 V=800.0 PL=0
MOVL C01310 V=800.0 PL=0
MOVL C01311 V=800.0 PL=0
MOVL C01312 V=800.0 PL=0
MOVL C01313 V=800.0 PL=0
MOVL C01314 V=800.0 PL=0
MOVL C01315 V=800.0 PL=0
MOVL C01316 V=800.0 PL=0
MOVL C01317 V=800.0 PL=0
MOVL C01318 V=800.0 PL=0
MOVL C01319 V=800.0 PL=0
MOVL C01320 V=800.0 PL=0
MOVL C01321 V=800.0 PL=0
MOVL C01322 V=800.0 PL=0
MOVL C01323 V=800.0 PL=0
MOVL C01324 V=800.0 PL=0
MOVL C01325 V=800.0 PL=0
MOVL C01326 V=800.0 PL=0
MOVL C01327 V=800.0 PL=0
MOVL C01328 V=800.0 PL=0
MOVL C01329 V=800.0 PL=0
MOVL C01330 V=800.0 PL=0
MOVL C01331 V=800.0 PL=0
MOVL C01332 V=800.0 PL=0
MOVL C01333 V=800.0 PL=0
MOVL C01334 V=800.0 PL=0
MOVL C01335 V=800.0 PL=0
MOVL C01336 V=800.0 PL=0
MOVL C01337 V=800.0 PL=0
MOVL C01338 V=800.0 PL=0
MOVL C01339 V=800.0 PL=0
MOVL C01340 V=800.0 PL=0
MOVL C01341 V=800.0 PL=0
MOVL C01342 V=800.0 PL=0
MOVL C01343 V=800.0 PL=0
MOVL C01344 V=800.0 PL=0
MOVL C01345 V=800.0 PL=0
MOVL C01346 V=800.0 PL=0
MOVL C01347 V=800.0 PL=0
MOVL C01348 V=800.0 PL=0
MOVL C01349 V=800.0 PL=0
MOVL C01350 V=800.0 PL=0
MOVL C01351 V=800.0 PL=0
MOVL C01352 V=800.0 PL=0
MOVL C01353 V=800.0 PL=0
MOVL C01354 V=800.0 PL=0
MOVL C01355 V=800.0 PL=0
MOVL C01356 V=800.0 PL=0
MOVL C01357 V=800.0 PL=0
MOVL C01358 V=800.0 PL=0
MOVL C01359 V=800.0 PL=0
MOVL C01360 V=800.0 PL=0
MOVL C01361 V=800.0 PL=0
MOVL C01362 V=800.0 PL=0
MOVL C01363 V=800.0 PL=0
MOVL C01364 V=800.0 PL=0
MOVL C01365 V=800.0 PL=0
MOVL C01366 V=800.0 PL=0
MOVL C01367 V=800.0 PL=0
MOVL C01368 V=800.0 PL=0
MOVL C01369 V=800.0 PL=0
MOVL C01370 V=800.0 PL=0
MOVL C01371 V=800.0 PL=0
MOVL C01372 V=800.0 PL=0
MOVL C01373 V=800.0 PL=0
MOVL C01374 V=800.0 PL=0
MOVL C01375 V=800.0 PL=0
MOVL C01376 V=800.0 PL=0
MOVL C01377 V=800.0 PL=0
MOVL C01378 V=800.0 PL=0
MOVL C01379 V=800.0 PL=0
MOVL C01380 V=800.0 PL=0
MOVL C01381 V=800.0 PL=0
MOVL C01382 V=800.0 PL=0
MOVL C01383 V=800.0 PL=0
MOVL C01384 V=800.0 PL=0
MOVL C01385 V=800.0 PL=0
MOVL C01386 V=800.0 PL=0
MOVL C01387 V=800.0 PL=0
MOVL C01388 V=800.0 PL=0
MOVL C01389 V=800.0 PL=0
MOVL C01390 V=800.0 PL=0
MOVL C01391 V=800.0 PL=0
MOVL C01392 V=800.0 PL=0
MOVL C01393 V=800.0 PL=0
MOVL C01394 V=800.0 PL=0
MOVL C01395 V=800.0 PL=0
MOVL C01396 V=800.0 PL=0
MOVL C01397 V=800.0 PL=0
MOVL C01398 V=800.0 PL=0
MOVL C01399 V=800.0 PL=0
MOVL C01400 V=800.0 PL=0
MOVL C01401 V=800.0 PL=0
MOVL C01402 V=800.0 PL=0
MOVL C01403 V=800.0 PL=0
MOVL C01404 V=800.0 PL=0
MOVL C01405 V=800.0 PL=0
MOVL C01406 V=800.0 PL=0
MOVL C01407 V=800.0 PL=0
MOVL C01408 V=800.0 PL=0
MOVL C01409 V=800.0 PL=0
MOVL C01410 V=800.0 PL=0
MOVL C01411 V=800.0 PL=0
MOVL C01412 V=800.0 PL=0
MOVL C01413 V=800.0 PL=0
MOVL C01414 V=800.0 PL=0
MOVL C01415 V=800.0 PL=0
MOVL C01416 V=800.0 PL=0
MOVL C01417 V=800.0 PL=0
MOVL C01418 V=800.0 PL=0
MOVL C01419 V=800.0 PL=0
MOVL C01420 V=800.0 PL=0
MOVL C01421 V=800.0 PL=0
MOVL C01422 V=800.0 PL=0
MOVL C01423 V=800.0 PL=0
MOVL C01424 V=800.0 PL=0
MOVL C01425 V=800.0 PL=0
MOVL C01426 V=800.0 PL=0
MOVL C01427 V=800.0 PL=0
MOVL C01428 V=800.0 PL=0
MOVL C01429 V=800.0 PL=0
MOVL C01430 V=800.0 PL=0
MOVL C01431 V=800.0 PL=0
MOVL C01432 V=800.0 PL=0
MOVL C01433 V=800.0 PL=0
MOVL C01434 V=800.0 PL=0
MOVL C01435 V=800.0 PL=0
MOVL C01436 V=800.0 PL=0
MOVL C01437 V=800.0 PL=0
MOVL C01438 V=800.0 PL=0
MOVL C01439 V=800.0 PL=0
MOVL C01440 V=800.0 PL=0
MOVL C01441 V=800.0 PL=0
MOVL C01442 V=800.0 PL=0
MOVL C01443 V=800.0 PL=0
MOVL C01444 V=800.0 PL=0
MOVL C01445 V=800.0 PL=0
MOVL C01446 V=800.0 PL=0
MOVL C01447 V=800.0 PL=0
MOVL C01448 V=800.0 PL=0
MOVL C01449 V=800.0 PL=0
MOVL C01450 V=800.0 PL=0
MOVL C01451 V=800.0 PL=0
MOVL C01452 V=800.0 PL=0
MOVL C01453 V=800.0 PL=0
MOVL C01454 V=800.0 PL=0
MOVL C01455 V=800.0 PL=0
MOVL C01456 V=800.0 PL=0
MOVL C01457 V=800.0 PL=0
MOVL C01458 V=800.0 PL=0
MOVL C01459 V=800.0 PL=0
MOVL C01460 V=800.0 PL=0
MOVL C01461 V=800.0 PL=0
MOVL C01462 V=800.0 PL=0
MOVL C01463 V=800.0 PL=0
MOVL C01464 V=800.0 PL=0
MOVL C01465 V=800.0 PL=0
MOVL C01466 V=800.0 PL=0
MOVL C01467 V=800.0 PL=0
MOVL C01468 V=800.0 PL=0
MOVL C01469 V=800.0 PL=0
MOVL C01470 V=800.0 PL=0
MOVL C01471 V=800.0 PL=0
MOVL C01472 V=800.0 PL=0
MOVL C01473 V=800.0 PL=0
MOVL C01474 V=800.0 PL=0
MOVL C01475 V=800.0 PL=0
MOVL C01476 V=800.0 PL=0
MOVL C01477 V=800.0 PL=0
MOVL C01478 V=800.0 PL=0
MOVL C01479 V=800.0 PL=0
MOVL C01480 V=800.0 PL=0
MOVL C01481 V=800.0 PL=0
MOVL C01482 V=800.0 PL=0
MOVL C01483 V=800.0 PL=0
MOVL C01484 V=800.0 PL=0
MOVL C01485 V=800.0 PL=0
MOVL C01486 V=800.0 PL=0
MOVL C01487 V=800.0 PL=0
MOVL C01488 V=800.0 PL=0
MOVL C01489 V=800.0 PL=0
MOVL C01490 V=800.0 PL=0
MOVL C01491 V=800.0 PL=0
MOVL C01492 V=800.0 PL=0
MOVL C01493 V=800.0 PL=0
MOVL C01494 V=800.0 PL=0
MOVL C01495 V=800.0 PL=0
MOVL C01496 V=800.0 PL=0
MOVL C01497 V=800.0 PL=0
MOVL C01498 V=800.0 PL=0
MOVL C01499 V=800.0 PL=0
MOVL C01500 V=800.0 PL=0
MOVL C01501 V=800.0 PL=0
MOVL C01502 V=800.0 PL=0
MOVL C01503 V=800.0 PL=0
MOVL C01504 V=800.0 PL=0
MOVL C01505 V=800.0 PL=0
MOVL C01506 V=800.0 PL=0
MOVL C01507 V=800.0 PL=0
MOVL C01508 V=800.0 PL=0
MOVL C01509 V=800.0 PL=0
MOVL C01510 V=800.0 PL=0
MOVL C01511 V=800.0 PL=0
MOVL C01512 V=800.0 PL=0
MOVL C01513 V=800.0 PL=0
MOVL C01514 V=800.0 PL=0
MOVL C01515 V=800.0 PL=0
MOVL C01516 V=800.0 PL=0
MOVL C01517 V=800.0 PL=0
MOVL C01518 V=800.0 PL=0
MOVL C01519 V=800.0 PL=0
MOVL C01520 V=800.0 PL=0
MOVL C01521 V=800.0 PL=0
MOVL C01522 V=800.0 PL=0
MOVL C01523 V=800.0 PL=0
MOVL C01524 V=800.0 PL=0
MOVL C01525 V=800.0 PL=0
MOVL C01526 V=800.0 PL=0
MOVL C01527 V=800.0 PL=0
MOVL C01528 V=800.0 PL=0
MOVL C01529 V=800.0 PL=0
MOVL C01530 V=800.0 PL=0
MOVL C01531 V=800.0 PL=0
MOVL C01532 V=800.0 PL=0
MOVL C01533 V=800.0 PL=0
MOVL C01534 V=800.0 PL=0
MOVL C01535 V=800.0 PL=0
MOVL C01536 V=800.0 PL=0
MOVL C01537 V=800.0 PL=0
MOVL C01538 V=800.0 PL=0
MOVL C01539 V=800.0 PL=0
MOVL C01540 V=800.0 PL=0
MOVL C01541 V=800.0 PL=0
MOVL C01542 V=800.0 PL=0
MOVL C01543 V=800.0 PL=0
MOVL C01544 V=800.0 PL=0
MOVL C01545 V=800.0 PL=0
MOVL C01546 V=800.0 PL=0
MOVL C01547 V=800.0 PL=0
MOVL C01548 V=800.0 PL=0
MOVL C01549 V=800.0 PL=0
MOVL C01550 V=800.0 PL=0
MOVL C01551 V=800.0 PL=0
MOVL C01552 V=800.0 PL=0
MOVL C01553 V=800.0 PL=0
MOVL C01554 V=800.0 PL=0
MOVL C01555 V=800.0 PL=0
MOVL C01556 V=800.0 PL=0
MOVL C01557 V=800.0 PL=0
MOVL C01558 V=800.0 PL=0
MOVL C01559 V=800.0 PL=0
MOVL C01560 V=800.0 PL=0
MOVL C01561 V=800.0 PL=0
MOVL C01562 V=800.0 PL=0
MOVL C01563 V=800.0 PL=0
MOVL C01564 V=800.0 PL=0
MOVL C01565 V=800.0 PL=0
MOVL C01566 V=800.0 PL=0
MOVL C01567 V=800.0 PL=0
MOVL C01568 V=800.0 PL=0
MOVL C01569 V=800.0 PL=0
MOVL C01570 V=800.0 PL=0
MOVL C01571 V=800.0 PL=0
MOVL C01572 V=800.0 PL=0
MOVL C01573 V=800.0 PL=0
MOVL C01574 V=800.0 PL=0
MOVL C01575 V=800.0 PL=0
MOVL C01576 V=800.0 PL=0
MOVL C01577 V=800.0 PL=0
MOVL C01578 V=800.0 PL=0
MOVL C01579 V=800.0 PL=0
MOVL C01580 V=800.0 PL=0
MOVL C01581 V=800.0 PL=0
MOVL C01582 V=800.0 PL=0
MOVL C01583 V=800.0 PL=0
MOVL C01584 V=800.0 PL=0
MOVL C01585 V=800.0 PL=0
MOVL C01586 V=800.0 PL=0
MOVL C01587 V=800.0 PL=0
MOVL C01588 V=800.0 PL=0
MOVL C01589 V=800.0 PL=0
MOVL C01590 V=800.0 PL=0
MOVL C01591 V=800.0 PL=0
MOVL C01592 V=800.0 PL=0
MOVL C01593 V=800.0 PL=0
MOVL C01594 V=800.0 PL=0
MOVL C01595 V=800.0 PL=0
MOVL C01596 V=800.0 PL=0
MOVL C01597 V=800.0 PL=0
MOVL C01598 V=800.0 PL=0
MOVL C01599 V=800.0 PL=0
MOVL C01600 V=800.0 PL=0
MOVL C01601 V=800.0 PL=0
MOVL C01602 V=800.0 PL=0
MOVL C01603 V=800.0 PL=0
MOVL C01604 V=800.0 PL=0
MOVL C01605 V=800.0 PL=0
MOVL C01606 V=800.0 PL=0
MOVL C01607 V=800.0 PL=0
MOVL C01608 V=800.0 PL=0
MOVL C01609 V=800.0 PL=0
MOVL C01610 V=800.0 PL=0
MOVL C01611 V=800.0 PL=0
MOVL C01612 V=800.0 PL=0
MOVL C01613 V=800.0 PL=0
MOVL C01614 V=800.0 PL=0
MOVL C01615 V=800.0 PL=0
MOVL C01616 V=800.0 PL=0
MOVL C01617 V=800.0 PL=0
MOVL C01618 V=800.0 PL=0
MOVL C01619 V=800.0 PL=0
MOVL C01620 V=800.0 PL=0
MOVL C01621 V=800.0 PL=0
MOVL C01622 V=800.0 PL=0
MOVL C01623 V=800.0 PL=0
MOVL C01624 V=800.0 PL=0
MOVL C01625 V=800.0 PL=0
MOVL C01626 V=800.0 PL=0
MOVL C01627 V=800.0 PL=0
MOVL C01628 V=800.0 PL=0
MOVL C01629 V=800.0 PL=0
MOVL C01630 V=800.0 PL=0
MOVL C01631 V=800.0 PL=0
MOVL C01632 V=800.0 PL=0
MOVL C01633 V=800.0 PL=0
MOVL C01634 V=800.0 PL=0
MOVL C01635 V=800.0 PL=0
MOVL C01636 V=800.0 PL=0
MOVL C01637 V=800.0 PL=0
MOVL C01638 V=800.0 PL=0
MOVL C01639 V=800.0 PL=0
MOVL C01640 V=800.0 PL=0
MOVL C01641 V=800.0 PL=0
MOVL C01642 V=800.0 PL=0
MOVL C01643 V=800.0 PL=0
MOVL C01644 V=800.0 PL=0
MOVL C01645 V=800.0 PL=0
MOVL C01646 V=800.0 PL=0
MOVL C01647 V=800.0 PL=0
MOVL C01648 V=800.0 PL=0
MOVL C01649 V=800.0 PL=0
MOVL C01650 V=800.0 PL=0
MOVL C01651 V=800.0 PL=0
MOVL C01652 V=800.0 PL=0
MOVL C01653 V=800.0 PL=0
MOVL C01654 V=800.0 PL=0
MOVL C01655 V=800.0 PL=0
MOVL C01656 V=800.0 PL=0
MOVL C01657 V=800.0 PL=0
MOVL C01658 V=800.0 PL=0
MOVL C01659 V=800.0 PL=0
MOVL C01660 V=800.0 PL=0
MOVL C01661 V=800.0 PL=0
MOVL C01662 V=800.0 PL=0
MOVL C01663 V=800.0 PL=0
MOVL C01664 V=800.0 PL=0
MOVL C01665 V=800.0 PL=0
MOVL C01666 V=800.0 PL=0
MOVL C01667 V=800.0 PL=0
MOVL C01668 V=800.0 PL=0
MOVL C01669 V=800.0 PL=0
MOVL C01670 V=800.0 PL=0
MOVL C01671 V=800.0 PL=0
MOVL C01672 V=800.0 PL=0
MOVL C01673 V=800.0 PL=0
MOVL C01674 V=800.0 PL=0
MOVL C01675 V=800.0 PL=0
MOVL C01676 V=800.0 PL=0
MOVL C01677 V=800.0 PL=0
MOVL C01678 V=800.0 PL=0
MOVL C01679 V=800.0 PL=0
MOVL C01680 V=800.0 PL=0
MOVL C01681 V=800.0 PL=0
MOVL C01682 V=800.0 PL=0
MOVL C01683 V=800.0 PL=0
MOVL C01684 V=800.0 PL=0
MOVL C01685 V=800.0 PL=0
MOVL C01686 V=800.0 PL=0
MOVL C01687 V=800.0 PL=0
MOVL C01688 V=800.0 PL=0
MOVL C01689 V=800.0 PL=0
MOVL C01690 V=800.0 PL=0
MOVL C01691 V=800.0 PL=0
MOVL C01692 V=800.0 PL=0
MOVL C01693 V=800.0 PL=0
MOVL C01694 V=800.0 PL=0
MOVL C01695 V=800.0 PL=0
MOVL C01696 V=800.0 PL=0
MOVL C01697 V=800.0 PL=0
MOVL C01698 V=800.0 PL=0
MOVL C01699 V=800.0 PL=0
MOVL C01700 V=800.0 PL=0
MOVL C01701 V=800.0 PL=0
MOVL C01702 V=800.0 PL=0
MOVL C01703 V=800.0 PL=0
MOVL C01704 V=800.0 PL=0
MOVL C01705 V=800.0 PL=0
MOVL C01706 V=800.0 PL=0
MOVL C01707 V=800.0 PL=0
MOVL C01708 V=800.0 PL=0
MOVL C01709 V=800.0 PL=0
MOVL C01710 V=800.0 PL=0
MOVL C01711 V=800.0 PL=0
MOVL C01712 V=800.0 PL=0
MOVL C01713 V=800.0 PL=0
MOVL C01714 V=800.0 PL=0
MOVL C01715 V=800.0 PL=0
MOVL C01716 V=800.0 PL=0
MOVL C01717 V=800.0 PL=0
MOVL C01718 V=800.0 PL=0
MOVL C01719 V=800.0 PL=0
MOVL C01720 V=800.0 PL=0
MOVL C01721 V=800.0 PL=0
MOVL C01722 V=800.0 PL=0
MOVL C01723 V=800.0 PL=0
MOVL C01724 V=800.0 PL=0
MOVL C01725 V=800.0 PL=0
MOVL C01726 V=800.0 PL=0
MOVL C01727 V=800.0 PL=0
MOVL C01728 V=800.0 PL=0
MOVL C01729 V=800.0 PL=0
MOVL C01730 V=800.0 PL=0
MOVL C01731 V=800.0 PL=0
MOVL C01732 V=800.0 PL=0
MOVL C01733 V=800.0 PL=0
MOVL C01734 V=800.0 PL=0
MOVL C01735 V=800.0 PL=0
MOVL C01736 V=800.0 PL=0
MOVL C01737 V=800.0 PL=0
MOVL C01738 V=800.0 PL=0
MOVL C01739 V=800.0 PL=0
MOVL C01740 V=800.0 PL=0
MOVL C01741 V=800.0 PL=0
MOVL C01742 V=800.0 PL=0
MOVL C01743 V=800.0 PL=0
MOVL C01744 V=800.0 PL=0
MOVL C01745 V=800.0 PL=0
MOVL C01746 V=800.0 PL=0
MOVL C01747 V=800.0 PL=0
MOVL C01748 V=800.0 PL=0
MOVL C01749 V=800.0 PL=0
MOVL C01750 V=800.0 PL=0
MOVL C01751 V=800.0 PL=0
MOVL C01752 V=800.0 PL=0
MOVL C01753 V=800.0 PL=0
MOVL C01754 V=800.0 PL=0
MOVL C01755 V=800.0 PL=0
MOVL C01756 V=800.0 PL=0
MOVL C01757 V=800.0 PL=0
MOVL C01758 V=800.0 PL=0
MOVL C01759 V=800.0 PL=0
MOVL C01760 V=800.0 PL=0
MOVL C01761 V=800.0 PL=0
MOVL C01762 V=800.0 PL=0
MOVL C01763 V=800.0 PL=0
MOVL C01764 V=800.0 PL=0
MOVL C01765 V=800.0 PL=0
MOVL C01766 V=800.0 PL=0
MOVL C01767 V=800.0 PL=0
MOVL C01768 V=800.0 PL=0
MOVL C01769 V=800.0 PL=0
MOVL C01770 V=800.0 PL=0
MOVL C01771 V=800.0 PL=0
MOVL C01772 V=800.0 PL=0
MOVL C01773 V=800.0 PL=0
MOVL C01774 V=800.0 PL=0
MOVL C01775 V=800.0 PL=0
MOVL C01776 V=800.0 PL=0
MOVL C01777 V=800.0 PL=0
MOVL C01778 V=800.0 PL=0
MOVL C01779 V=800.0 PL=0
MOVL C01780 V=800.0 PL=0
MOVL C01781 V=800.0 PL=0
MOVL C01782 V=800.0 PL=0
MOVL C01783 V=800.0 PL=0
MOVL C01784 V=800.0 PL=0
MOVL C01785 V=800.0 PL=0
MOVL C01786 V=800.0 PL=0
MOVL C01787 V=800.0 PL=0
MOVL C01788 V=800.0 PL=0
MOVL C01789 V=800.0 PL=0
MOVL C01790 V=800.0 PL=0
MOVL C01791 V=800.0 PL=0
MOVL C01792 V=800.0 PL=0
MOVL C01793 V=800.0 PL=0
MOVL C01794 V=800.0 PL=0
MOVL C01795 V=800.0 PL=0
MOVL C01796 V=800.0 PL=0
MOVL C01797 V=800.0 PL=0
MOVL C01798 V=800.0 PL=0
MOVL C01799 V=800.0 PL=0
MOVL C01800 V=800.0 PL=0
MOVL C01801 V=800.0 PL=0
MOVL C01802 V=800.0 PL=0
MOVL C01803 V=800.0 PL=0
MOVL C01804 V=800.0 PL=0
MOVL C01805 V=800.0 PL=0
MOVL C01806 V=800.0 PL=0
MOVL C01807 V=800.0 PL=0
MOVL C01808 V=800.0 PL=0
MOVL C01809 V=800.0 PL=0
MOVL C01810 V=800.0 PL=0
MOVL C01811 V=800.0 PL=0
MOVL C01812 V=800.0 PL=0
MOVL C01813 V=800.0 PL=0
MOVL C01814 V=800.0 PL=0
MOVL C01815 V=800.0 PL=0
MOVL C01816 V=800.0 PL=0
MOVL C01817 V=800.0 PL=0
MOVL C01818 V=800.0 PL=0
MOVL C01819 V=800.0 PL=0
MOVL C01820 V=800.0 PL=0
MOVL C01821 V=800.0 PL=0
MOVL C01822 V=800.0 PL=0
MOVL C01823 V=800.0 PL=0
MOVL C01824 V=800.0 PL=0
MOVL C01825 V=800.0 PL=0
MOVL C01826 V=800.0 PL=0
MOVL C01827 V=800.0 PL=0
MOVL C01828 V=800.0 PL=0
MOVL C01829 V=800.0 PL=0
MOVL C01830 V=800.0 PL=0
MOVL C01831 V=800.0 PL=0
MOVL C01832 V=800.0 PL=0
MOVL C01833 V=800.0 PL=0
MOVL C01834 V=800.0 PL=0
MOVL C01835 V=800.0 PL=0
MOVL C01836 V=800.0 PL=0
MOVL C01837 V=800.0 PL=0
MOVL C01838 V=800.0 PL=0
MOVL C01839 V=800.0 PL=0
MOVL C01840 V=800.0 PL=0
MOVL C01841 V=800.0 PL=0
MOVL C01842 V=800.0 PL=0
MOVL C01843 V=800.0 PL=0
MOVL C01844 V=800.0 PL=0
MOVL C01845 V=800.0 PL=0
MOVL C01846 V=800.0 PL=0
MOVL C01847 V=800.0 PL=0
MOVL C01848 V=800.0 PL=0
MOVL C01849 V=800.0 PL=0
MOVL C01850 V=800.0 PL=0
MOVL C01851 V=800.0 PL=0
MOVL C01852 V=800.0 PL=0
MOVL C01853 V=800.0 PL=0
MOVL C01854 V=800.0 PL=0
MOVL C01855 V=800.0 PL=0
MOVL C01856 V=800.0 PL=0
MOVL C01857 V=800.0 PL=0
MOVL C01858 V=800.0 PL=0
MOVL C01859 V=800.0 PL=0
MOVL C01860 V=800.0 PL=0
MOVL C01861 V=800.0 PL=0
MOVL C01862 V=800.0 PL=0
MOVL C01863 V=800.0 PL=0
MOVL C01864 V=800.0 PL=0
MOVL C01865 V=800.0 PL=0
MOVL C01866 V=800.0 PL=0
MOVL C01867 V=800.0 PL=0
MOVL C01868 V=800.0 PL=0
MOVL C01869 V=800.0 PL=0
MOVL C01870 V=800.0 PL=0
MOVL C01871 V=800.0 PL=0
MOVL C01872 V=800.0 PL=0
MOVL C01873 V=800.0 PL=0
MOVL C01874 V=800.0 PL=0
MOVL C01875 V=800.0 PL=0
MOVL C01876 V=800.0 PL=0
MOVL C01877 V=800.0 PL=0
MOVL C01878 V=800.0 PL=0
MOVL C01879 V=800.0 PL=0
MOVL C01880 V=800.0 PL=0
MOVL C01881 V=800.0 PL=0
MOVL C01882 V=800.0 PL=0
MOVL C01883 V=800.0 PL=0
MOVL C01884 V=800.0 PL=0
MOVL C01885 V=800.0 PL=0
MOVL C01886 V=800.0 PL=0
MOVL C01887 V=800.0 PL=0
MOVL C01888 V=800.0 PL=0
MOVL C01889 V=800.0 PL=0
MOVL C01890 V=800.0 PL=0
MOVL C01891 V=800.0 PL=0
MOVL C01892 V=800.0 PL=0
MOVL C01893 V=800.0 PL=0
MOVL C01894 V=800.0 PL=0
MOVL C01895 V=800.0 PL=0
MOVL C01896 V=800.0 PL=0
MOVL C01897 V=800.0 PL=0
MOVL C01898 V=800.0 PL=0
MOVL C01899 V=800.0 PL=0
MOVL C01900 V=800.0 PL=0
MOVL C01901 V=800.0 PL=0
MOVL C01902 V=800.0 PL=0
MOVL C01903 V=800.0 PL=0
MOVL C01904 V=800.0 PL=0
MOVL C01905 V=800.0 PL=0
MOVL C01906 V=800.0 PL=0
MOVL C01907 V=800.0 PL=0
MOVL C01908 V=800.0 PL=0
MOVL C01909 V=800.0 PL=0
MOVL C01910 V=800.0 PL=0
MOVL C01911 V=800.0 PL=0
MOVL C01912 V=800.0 PL=0
MOVL C01913 V=800.0 PL=0
MOVL C01914 V=800.0 PL=0
MOVL C01915 V=800.0 PL=0
MOVL C01916 V=800.0 PL=0
MOVL C01917 V=800.0 PL=0
MOVL C01918 V=800.0 PL=0
MOVL C01919 V=800.0 PL=0
MOVL C01920 V=800.0 PL=0
MOVL C01921 V=800.0 PL=0
MOVL C01922 V=800.0 PL=0
MOVL C01923 V=800.0 PL=0
MOVL C01924 V=800.0 PL=0
MOVL C01925 V=800.0 PL=0
MOVL C01926 V=800.0 PL=0
MOVL C01927 V=800.0 PL=0
MOVL C01928 V=800.0 PL=0
MOVL C01929 V=800.0 PL=0
MOVL C01930 V=800.0 PL=0
MOVL C01931 V=800.0 PL=0
MOVL C01932 V=800.0 PL=0
MOVL C01933 V=800.0 PL=0
MOVL C01934 V=800.0 PL=0
MOVL C01935 V=800.0 PL=0
MOVL C01936 V=800.0 PL=0
MOVL C01937 V=800.0 PL=0
MOVL C01938 V=800.0 PL=0
MOVL C01939 V=800.0 PL=0
MOVL C01940 V=800.0 PL=0
MOVL C01941 V=800.0 PL=0
MOVL C01942 V=800.0 PL=0
MOVL C01943 V=800.0 PL=0
MOVL C01944 V=800.0 PL=0
MOVL C01945 V=800.0 PL=0
MOVL C01946 V=800.0 PL=0
MOVL C01947 V=800.0 PL=0
MOVL C01948 V=800.0 PL=0
MOVL C01949 V=800.0 PL=0
MOVL C01950 V=800.0 PL=0
MOVL C01951 V=800.0 PL=0
MOVL C01952 V=800.0 PL=0
MOVL C01953 V=800.0 PL=0
MOVL C01954 V=800.0 PL=0
MOVL C01955 V=800.0 PL=0
MOVL C01956 V=800.0 PL=0
MOVL C01957 V=800.0 PL=0
MOVL C01958 V=800.0 PL=0
MOVL C01959 V=800.0 PL=0
MOVL C01960 V=800.0 PL=0
MOVL C01961 V=800.0 PL=0
MOVL C01962 V=800.0 PL=0
MOVL C01963 V=800.0 PL=0
MOVL C01964 V=800.0 PL=0
MOVL C01965 V=800.0 PL=0
MOVL C01966 V=800.0 PL=0
MOVL C01967 V=800.0 PL=0
MOVL C01968 V=800.0 PL=0
MOVL C01969 V=800.0 PL=0
MOVL C01970 V=800.0 PL=0
MOVL C01971 V=800.0 PL=0
MOVL C01972 V=800.0 PL=0
MOVL C01973 V=800.0 PL=0
MOVL C01974 V=800.0 PL=0
MOVL C01975 V=800.0 PL=0
MOVL C01976 V=800.0 PL=0
MOVL C01977 V=800.0 PL=0
MOVL C01978 V=800.0 PL=0
MOVL C01979 V=800.0 PL=0
MOVL C01980 V=800.0 PL=0
MOVL C01981 V=800.0 PL=0
MOVL C01982 V=800.0 PL=0
MOVL C01983 V=800.0 PL=0
MOVL C01984 V=800.0 PL=0
MOVL C01985 V=800.0 PL=0
MOVL C01986 V=800.0 PL=0
MOVL C01987 V=800.0 PL=0
MOVL C01988 V=800.0 PL=0
MOVL C01989 V=800.0 PL=0
MOVL C01990 V=800.0 PL=0
MOVL C01991 V=800.0 PL=0
MOVL C01992 V=800.0 PL=0
MOVL C01993 V=800.0 PL=0
MOVL C01994 V=800.0 PL=0
MOVL C01995 V=800.0 PL=0
MOVL C01996 V=800.0 PL=0
MOVL C01997 V=800.0 PL=0
MOVL C01998 V=800.0 PL=0
MOVL C01999 V=800.0 PL=0
MOVL C02000 V=800.0 PL=0
MOVL C02001 V=800.0 PL=0
MOVL C02002 V=800.0 PL=0
MOVL C02003 V=800.0 PL=0
MOVL C02004 V=800.0 PL=0
MOVL C02005 V=800.0 PL=0
MOVL C02006 V=800.0 PL=0
MOVL C02007 V=800.0 PL=0
MOVL C02008 V=800.0 PL=0
MOVL C02009 V=800.0 PL=0
MOVL C02010 V=800.0 PL=0
MOVL C02011 V=800.0 PL=0
MOVL C02012 V=800.0 PL=0
MOVL C02013 V=800.0 PL=0
MOVL C02014 V=800.0 PL=0
MOVL C02015 V=800.0 PL=0
MOVL C02016 V=800.0 PL=0
MOVL C02017 V=800.0 PL=0
MOVL C02018 V=800.0 PL=0
MOVL C02019 V=800.0 PL=0
MOVL C02020 V=800.0 PL=0
MOVL C02021 V=800.0 PL=0
MOVL C02022 V=800.0 PL=0
MOVL C02023 V=800.0 PL=0
MOVL C02024 V=800.0 PL=0
MOVL C02025 V=800.0 PL=0
MOVL C02026 V=800.0 PL=0
MOVL C02027 V=800.0 PL=0
MOVL C02028 V=800.0 PL=0
MOVL C02029 V=800.0 PL=0
MOVL C02030 V=800.0 PL=0
MOVL C02031 V=800.0 PL=0
MOVL C02032 V=800.0 PL=0
MOVL C02033 V=800.0 PL=0
MOVL C02034 V=800.0 PL=0
MOVL C02035 V=800.0 PL=0
